// TIA Portal V20 program export: 15 tag tables, 106 data types, 49 data blocks, 136 code blocks (in call order from the OBs), 146 instance data blocks

VAR_GLOBAL   // PLC tag table "Analog_Inputs"
   AI_LaserPowerMeter AT %IW412 : Word;
   AI_AxisB_ClampingPart AT %IW414 : Word;
   AI_LaserAirPressureProcess AT %IW416 : Word;
   AI_InletAirPressure AT %IW418 : Word;
   AI_AmbiantTemperature AT %IW428 : Word;
   AI_MachineTemperature AT %IW430 : Word;
   AI_ColdWaterTemperatureInput AT %IW432 : Word;
   AI_ColdWaterTemperatureOutput AT %IW434 : Word;
   AI_X_AxisTemperaturePT1000 AT %IW436 : Word;
   AI_Y_AxisTemperaturePT1000 AT %IW438 : Word;
   "AI_X_ AxisTemperaturePTC" AT %IW440 : Word;
   "AI_Y_ AxisTemperaturePTC" AT %IW442 : Word;
   AI_NozzleOverpressure AT %IW444 : Word;
   AI_OpticalPathOverpressure AT %IW446 : Word;
   AI_LaserHeadOverpressure AT %IW448 : Word;
   AI_ZL_AxisOverpressure AT %IW450 : Word;
   AI_XY_AxisOverpressure AT %IW452 : Word;
   AI_LeftAspiration AT %IW454 : Word;
   AI_RightAspiration AT %IW456 : Word;
   AI_FreeIW458 AT %IW458 : Word;
   AI_ClimTemperature AT %IW480 : Word;
   AI_FreeIW482 AT %IW482 : Word;
   AI_FreeIW484 AT %IW484 : Word;
   AI_FreeIW486 AT %IW486 : Word;
   AI_SensorControllerStation1 AT %IW460 : Word;
   AI_CabinetTemperature AT %IW462 : Word;
   AI_FreeIW464 AT %IW464 : Word;
   AI_FreeIW466 AT %IW466 : Word;
END_VAR

VAR_GLOBAL   // PLC tag table "Analog_Outputs"
   AQ_NozzleOverpressureSetPoint AT %QW428 : Word;
   AQ_FreeQW482 AT %QW430 : Word;
   AQ_VentilatorSetPoint AT %QW432 : Word;
   AQ_PropValveClimSetPoint AT %QW434 : Word;
END_VAR

VAR_GLOBAL   // PLC tag table "BW_Inputs"
   AI_LifeFlag AT %IW500 : Int;
   DI_JobDone AT %I502.0 : Bool;
   DI_LockShuttle AT %I504.0 : Bool;
   AI_DataSend AT %IW506 : Int;
   AI_DataReceive AT %IW508 : Int;
   DI_NoEmergencyStopAtBwLoader AT %I510.0 : Bool;
   DI_SafetyDoorsClosedAtBwLoader AT %I512.0 : Bool;
   AI_BwInErrorState AT %IW514 : Int;
   DI_UndrilledPartControl AT %I516.0 : Bool;
   DI_DrilledPartControl AT %I518.0 : Bool;
   DI_BackwallControl AT %I520.0 : Bool;
   DI_BwLoaderInSafePos AT %I522.0 : Bool;
   DI_SemiAutoValid AT %I562.0 : Bool;
END_VAR

VAR_GLOBAL   // PLC tag table "BW_Output"
   AQ_LifeFlag AT %QW500 : Int;
   DQ_LoaderRequest AT %Q502.0 : Bool;
   DQ_LockShuttle AT %Q504.0 : Bool;
   AQ_DataSend AT %QW506 : Int;
   AQ_DataReceive AT %QW508 : Int;
   DQ_NoEmergencyStopAtFemto AT %Q510.0 : Bool;
   DQ_SafetyDoorsClosedAtFemto AT %Q512.0 : Bool;
   AQ_FemtoInErrorState AT %QW514 : Int;
   DQ_AutoMode AT %Q516.0 : Bool;
   DQ_JogMode AT %Q518.0 : Bool;
   DQ_GotoSafePos AT %Q520.0 : Bool;
   AQ_Reset AT %QW526 : Int;
   DQ_Emptying AT %Q522.0 : Bool;
   DQ_BW_CtrlInProgress AT %Q524.0 : Bool;
END_VAR

VAR_GLOBAL   // PLC tag table "Cognex"
   ASTriggerReady AT %I690.0 : Bool;   // Acquisition status
   ASTriggerAck AT %I690.1 : Bool;   // Acquisition status
   ASAcquiring AT %I690.2 : Bool;   // Acquisition status
   ASMissedTrig AT %I690.3 : Bool;   // Acquisition status
   ASOfflineResBit1 AT %I690.4 : Bool;   // Acquisition status
   ASOfflineResBit2 AT %I690.5 : Bool;   // Acquisition status
   ASOfflineResBit3 AT %I690.6 : Bool;   // Acquisition status
   ASOnline AT %I690.7 : Bool;   // Acquisition status
   ASAcquiNum AT %IW691 : Word;   // Acquisition status
   ISInspecting AT %I693.0 : Bool;   // Inspection status
   ISToggleInspectDone AT %I693.1 : Bool;   // Inspection status
   ISBufferOverrun AT %I693.2 : Bool;   // Inspection status
   ISResultsValid AT %I693.3 : Bool;   // Inspection status
   ISJobLoading AT %I693.4 : Bool;   // Inspection status
   ISJobLoadComplete AT %I693.5 : Bool;   // Inspection status
   ISJobLoadFailed AT %I693.6 : Bool;   // Inspection status
   ISSetUserDataACk AT %I693.7 : Bool;   // Inspection status
   ISJobPass AT %I694.0 : Bool;   // Inspection status
   SEC0Ack AT %I699.0 : Bool;   // Soft event control
   SEC1Ack AT %I699.1 : Bool;   // Soft event control
   SEC2Ack AT %I699.2 : Bool;   // Soft event control
   SEC3Ack AT %I699.3 : Bool;   // Soft event control
   SEC4Ack AT %I699.4 : Bool;   // Soft event control
   SEC5Ack AT %I699.5 : Bool;   // Soft event control
   SEC6Ack AT %I699.6 : Bool;   // Soft event control
   SEC7Ack AT %I699.7 : Bool;   // Soft event control
   JCJobID AT %IW697 : Word;   // Job control
   IRInspectionID AT %IW600 : Word;   // Inspection result
   IRInspectResultCode AT %IW602 : Word;   // Inspection result
   IRActHoleNrResult AT %IB606 : Byte;   // Inspection result
   ResultDataFromCognex0 AT %ID604 : DWord;
   ResultDataFromCognex1 AT %ID608 : DWord;
   ResultDataFromCognex2 AT %ID612 : DWord;
   ResultDataFromCognex3 AT %ID616 : DWord;
   ACTriggerEnable AT %Q690.0 : Bool;   // Acquisition control
   ACTrigger AT %Q690.1 : Bool;   // Acquisition control
   ACClearAcquirCompl AT %Q690.2 : Bool;   // Acquisition control
   ACSetOffline AT %Q690.7 : Bool;   // Acquisition control
   ICBufferResultsEn AT %Q691.0 : Bool;   // Inspection control
   ICInspectResultsAck AT %Q691.1 : Bool;   // Inspection control
   ICSetUserData AT %Q691.2 : Bool;   // Inspection control
   ICExecuteCmd AT %Q691.3 : Bool;   // Inspection control
   CCSetJobID AT %QW697 : Word;   // Command control
   SEC0 AT %Q699.0 : Bool;   // Soft event control
   SEC1 AT %Q699.1 : Bool;   // Soft event control
   SEC2 AT %Q699.2 : Bool;   // Soft event control
   SEC3 AT %Q699.3 : Bool;   // Soft event control
   SEC4 AT %Q699.4 : Bool;   // Soft event control
   SEC5 AT %Q699.5 : Bool;   // Soft event control
   SEC6 AT %Q699.6 : Bool;   // Soft event control
   SEC7 AT %Q699.7 : Bool;   // Soft event control
   UserDataToCognex0 AT %QD600 : DWord;
   UserDataToCognex1 AT %QD604 : DWord;
   UserDataToCognex2 AT %QD608 : DWord;
   UserDataToCognex3 AT %QD612 : DWord;
   UserDataToCognex4 AT %QD616 : DWord;
   UserDataToCognex5 AT %QD620 : DWord;
   UserDataToCognex6 AT %QD624 : DWord;
   UserDataToCognex7 AT %QD628 : DWord;
END_VAR

VAR_GLOBAL   // PLC tag table "Default tag table"
   System_Byte AT %MB1 : Byte;
   FirstScan AT %M1.0 : Bool;
   DiagStatusUpdate AT %M1.1 : Bool;
   AlwaysTRUE AT %M1.2 : Bool;
   AlwaysFALSE AT %M1.3 : Bool;
   Clock_Byte AT %MB0 : Byte;
   Clock_10Hz AT %M0.0 : Bool;
   Clock_5Hz AT %M0.1 : Bool;
   "Clock_2.5Hz" AT %M0.2 : Bool;
   Clock_2Hz AT %M0.3 : Bool;
   "Clock_1.25Hz" AT %M0.4 : Bool;
   Clock_1Hz AT %M0.5 : Bool;
   "Clock_0.625Hz" AT %M0.6 : Bool;
   "Clock_0.5Hz" AT %M0.7 : Bool;
   Tag_1 AT %M99.0 : Bool;
   Tag_2 AT %MD1000 : DWord;
   Tag_3 AT %MW20 : Word;
   Tag_4 AT %MW40 : Word;
   Tag_5 AT %MW42 : Word;
   Tag_6 AT %MW44 : Word;
   Tag_7 AT %MW100 : Word;
   Tag_8 AT %MW102 : Word;
   Tag_9 AT %MW104 : Word;
   Tag_10 AT %MD150 : DWord;
END_VAR

VAR_GLOBAL   // PLC tag table "Digital_Inputs"
   DI_FreeI0_0 AT %I0.0 : Bool;
   DI_X_AxisBrakePressCtrl AT %I0.1 : Bool;
   DI_Y_AxisBrakePressCtrl AT %I0.2 : Bool;
   DI_BreakerCtrl AT %I0.3 : Bool;
   DI_CabinetTemperatureCtrl AT %I0.4 : Bool;
   DI_UPS_PowerFailure AT %I0.5 : Bool;
   DI_AirPressureCtrl AT %I0.6 : Bool;
   DI_ShutterClosed AT %I0.7 : Bool;
   DI_AirDryerOK AT %I1.0 : Bool;
   DI_UPS_BatteryOK AT %I1.1 : Bool;
   DI_FrontDoorClosed AT %I1.2 : Bool;
   DI_InfeedReadyOK_Start AT %I1.3 : Bool;
   DI_CoolingOK AT %I1.4 : Bool;
   DI_FreeI1_5 AT %I1.5 : Bool;
   DI_PowerReady AT %I1.6 : Bool;
   DI_AlarmI2T AT %I1.7 : Bool;
   DI_HeadLaserBusy AT %I2.0 : Bool;
   DI_HeadLaserBreaker AT %I2.1 : Bool;
   DI_FrontDoorLocked AT %I2.2 : Bool;
   DI_UPS_CommonAlarm AT %I2.3 : Bool;
   DI_UPS_BatteryLow AT %I2.4 : Bool;
   DI_FreeI2_5 AT %I2.5 : Bool;
   DI_HeadChillerHighPressure AT %I2.6 : Bool;
   DI_HeadChillerWaterTemperature AT %I2.7 : Bool;
   DI_HeadChillerFlow AT %I3.0 : Bool;
   DI_HeadChillerCollectivFault AT %I3.1 : Bool;
   DI_HeadChillerWaterLevel AT %I3.2 : Bool;
   DI_UPSByPassActive AT %I3.3 : Bool;
   DI_HeadChillerAmbiantTemperature AT %I3.4 : Bool;
   DI_FreeI3_5 AT %I3.5 : Bool;
   DI_FreeI3_6 AT %I3.6 : Bool;
   DI_FreeI3_7 AT %I3.7 : Bool;
   DI_LoadClampOpened AT %I4.0 : Bool;
   DI_LoadClampNotClosedWithPart AT %I4.1 : Bool;
   DI_UnloadClampOpened AT %I4.2 : Bool;
   DI_UPS_Fault AT %I4.3 : Bool;
   DI_InternalGateLocked AT %I4.4 : Bool;
   DI_ExternalGateLocked AT %I4.5 : Bool;
   DI_InverterActive AT %I4.6 : Bool;
   DI_UnloadClampNotClosedWithPart AT %I4.7 : Bool;
   DI_FreeI5_0 AT %I5.0 : Bool;
   DI_FreeI5_1 AT %I5.1 : Bool;
   DI_InternalGateOpened AT %I5.2 : Bool;
   DI_ExternalGateOpened AT %I5.3 : Bool;
   DI_PowerMeterBackCtrl AT %I5.4 : Bool;
   DI_PowerMeterFrontCtrl AT %I5.5 : Bool;
   DI_FreeI5_6 AT %I5.6 : Bool;
   DI_FreeI5_7 AT %I5.7 : Bool;
   DI_HeadChillerCutOff AT %I6.0 : Bool;
   DI_HeadChillerTemperature AT %I6.1 : Bool;
   DI_FreeI6_2 AT %I6.2 : Bool;
   DI_FreeI6_3 AT %I6.3 : Bool;
   DI_ClampingOpenCtrl AT %I6.4 : Bool;
   DI_B_AxisBrakeReleasedCtrl AT %I6.5 : Bool;
   "DI_FreeI6.6" AT %I6.6 : Bool;
   DI_B_AxisReferencePoint AT %I6.7 : Bool;
   DI_SourceChillerHighPressure AT %I7.0 : Bool;
   DI_SourceChillerWaterTemperature AT %I7.1 : Bool;
   DI_SourceChillerFlow AT %I7.2 : Bool;
   DI_SourceChillerCollectivFault AT %I7.3 : Bool;
   DI_SourceChillerWaterLevel AT %I7.4 : Bool;
   DI_SourceChillerAmbiantTemperature AT %I7.5 : Bool;
   DI_SourceChillerCutOff AT %I7.6 : Bool;
   DI_SourceChillerTemperature AT %I7.7 : Bool;
END_VAR

VAR_GLOBAL   // PLC tag table "Digital_Outputs"
   DQ_FreeQ0_0 AT %Q0.0 : Bool;
   DQ_OperatingCounter AT %Q0.1 : Bool;
   DQ_GeneralAirValve AT %Q0.2 : Bool;
   DQ_SmartLineDisable AT %Q0.3 : Bool;
   DQ_MachineLight AT %Q0.4 : Bool;
   DQ_MachineLightBack AT %Q0.5 : Bool;
   DQ_LightTowerOrange AT %Q0.6 : Bool;
   DQ_LightTowerRed AT %Q0.7 : Bool;
   DQ_LightTowerBlue AT %Q1.0 : Bool;
   DQ_Light_owerGreen AT %Q1.1 : Bool;
   DQ_LightTowerWhite AT %Q1.2 : Bool;
   DQ_Backlight AT %Q1.3 : Bool;
   DQ_FreeQ1_4 AT %Q1.4 : Bool;
   DQ_InfeedON AT %Q1.5 : Bool;
   DQ_AxisActivation AT %Q1.6 : Bool;
   DQ_BuzzerActivation AT %Q1.7 : Bool;
   DQ_ElbaronPowerON AT %Q2.0 : Bool;
   DQ_ObservationCameraLight AT %Q2.1 : Bool;
   DQ_LaserExternalDoorOpening AT %Q2.2 : Bool;
   DQ_CoolingStart AT %Q2.3 : Bool;
   DQ_X_AxisBrakeActivation AT %Q2.4 : Bool;
   DQ_Y_AxisBrakeActivation AT %Q2.5 : Bool;
   DQ_AxisB_TeachInClampingPart AT %Q2.6 : Bool;
   DQ_EPO_UPS AT %Q2.7 : Bool;
   DQ_HeadLaserStart AT %Q3.0 : Bool;
   DQ_HeadLaserStop AT %Q3.1 : Bool;
   DQ_Axis2_PowerContactor AT %Q3.2 : Bool;
   DQ_GasAssistOn AT %Q3.3 : Bool;
   DQ_SmartLineReset AT %Q3.4 : Bool;
   DQ_XY_AxisPowerContactor AT %Q3.5 : Bool;
   DQ_LaserAirPressureProcess AT %Q3.6 : Bool;
   DQ_Bus60V_PowerContactor AT %Q3.7 : Bool;
   DQ_FreeQ4_0 AT %Q4.0 : Bool;
   DQ_FreeQ4_1 AT %Q4.1 : Bool;
   DQ_FreeQ4_2 AT %Q4.2 : Bool;
   DQ_FreeQ4_3 AT %Q4.3 : Bool;
   DQ_LoadClampClosing AT %Q4.4 : Bool;
   DQ_LoadClampOpening AT %Q4.5 : Bool;
   DQ_UnloadClampClosing AT %Q4.6 : Bool;
   DQ_UnloadClampOpening AT %Q4.7 : Bool;
   DQ_ClampingOpening AT %Q5.0 : Bool;
   DQ_ClampingClosing AT %Q5.1 : Bool;
   DQ_B_AxisBrakeRelease AT %Q5.2 : Bool;
   DQ_Suction AT %Q5.3 : Bool;
   DQ_FreeQ5_4 AT %Q5.4 : Bool;
   DQ_FreeQ5_5 AT %Q5.5 : Bool;
   DQ_FreeQ5_6 AT %Q5.6 : Bool;
   DQ_FreeQ5_7 AT %Q5.7 : Bool;
   DQ_ExternalGateClosing AT %Q8.0 : Bool;
   DQ_ExternalGateOpening AT %Q8.1 : Bool;
   DQ_InternalGateClosing AT %Q8.2 : Bool;
   DQ_InternalGateOpening AT %Q8.3 : Bool;
   DQ_PowerMeterRetract AT %Q8.4 : Bool;
   DQ_PowerMeterAdvance AT %Q8.5 : Bool;
   DQ_Blowing AT %Q8.6 : Bool;   //    {ExternalWritable false}
   DQ_FreeQ8_7 AT %Q8.7 : Bool;
   DQ_FreeQ9_0 AT %Q9.0 : Bool;
   DQ_FreeQ9_1 AT %Q9.1 : Bool;
   DQ_FreeQ9_2 AT %Q9.2 : Bool;
   DQ_FreeQ9_3 AT %Q9.3 : Bool;
   DQ_FreeQ9_4 AT %Q9.4 : Bool;
   DQ_FreeQ9_5 AT %Q9.5 : Bool;
   DQ_FreeQ9_6 AT %Q9.6 : Bool;
   DQ_FreeQ9_7 AT %Q9.7 : Bool;
END_VAR

VAR_GLOBAL   // PLC tag table "F-Digital_Inputs"
   FDI_EStopCh1 AT %I1000.0 : Bool;
   FDI_KeySettingModeCh1 AT %I1000.1 : Bool;
   FDI_KeySettingLaserCh1 AT %I1000.2 : Bool;
   FDI_EStopFeedback AT %I1000.3 : Bool;
   FDI_EStopCh2 AT %I1000.4 : Bool;
   FDI_KeySettingModeCh2 AT %I1000.5 : Bool;
   FDI_KeySettingLaserCh2 AT %I1000.6 : Bool;
   FDI_ExternalFeedback AT %I1000.7 : Bool;
   FDI_ReturnPowerLaser AT %I1008.0 : Bool;
   FDI_MaintenanceDoorClosedCh1 AT %I1008.1 : Bool;
   FDI_FrontDoorClosedCh1 AT %I1008.2 : Bool;
   FDI_EstopPowerLaserCh1 AT %I1008.3 : Bool;
   FDI_ReturnShutterLaser AT %I1008.4 : Bool;
   FDI_MaintenanceDoorClosedCh2 AT %I1008.5 : Bool;
   FDI_FrontDoorClosedCh2 AT %I1008.6 : Bool;
   FDI_EstopPowerLaserCh2 AT %I1008.7 : Bool;
   FDI_RoofLeftDoorClosedCh1 AT %I1016.0 : Bool;
   FDI_LaserKeyON_Ch1 AT %I1016.1 : Bool;
   FDI_LaserExternalDoorClosedCh1 AT %I1016.2 : Bool;
   FDI_IntOrExtSasGatesClosedCh1 AT %I1016.3 : Bool;
   FDI_RoofLeftDoorClosedCh2 AT %I1016.4 : Bool;
   FDI_LaserKeyON_Ch2 AT %I1016.5 : Bool;
   FDI_LaserExternalDoorClosedCh2 AT %I1016.6 : Bool;
   FDI_IntOrExtSasGatesClosedCh2 AT %I1016.7 : Bool;
   FDI_BW_LoaderDoorClosedCh1 AT %I1024.0 : Bool;
   FDI_RoofRightDoorClosedCh1 AT %I1024.1 : Bool;
   FDI_SonplasEstopCh1 AT %I1024.2 : Bool;
   FDI_BW_LoaderEStopCh1 AT %I1024.3 : Bool;
   FDI_BW_LoaderDoorClosedCh2 AT %I1024.4 : Bool;
   FDI_RoofRightDoorClosedCh2 AT %I1024.5 : Bool;
   FDI_SonplasEstopCh2 AT %I1024.6 : Bool;
   FDI_BW_LoaderEStopCh2 AT %I1024.7 : Bool;
   FDI_SonplasDoorClosedCh1 AT %I1032.0 : Bool;
   FDI_FreeI1032_1 AT %I1032.1 : Bool;
   FDI_FreeI1032_2 AT %I1032.2 : Bool;
   FDI_FreeI1032_3 AT %I1032.3 : Bool;
   FDI_SonplasDoorClosedCh2 AT %I1032.4 : Bool;
   FDI_FreeI1032_5 AT %I1032.5 : Bool;
   FDI_FreeI1032_6 AT %I1032.6 : Bool;
   FDI_DoorClosedFeedback AT %I1032.7 : Bool;
END_VAR

VAR_GLOBAL   // PLC tag table "F-Digital_Outputs"
   FDQ_StopContactor AT %Q1200.0 : Bool;
   FDQ_LaserContactor AT %Q1200.1 : Bool;
   FDQ_LaserValidation AT %Q1200.2 : Bool;
   FDQ_FrontDoorLock AT %Q1200.3 : Bool;
   FDQ_BW_LoaderEstopRelay AT %Q1206.0 : Bool;
   FDQ_SonplasDoorClosedRelay AT %Q1206.1 : Bool;
   FDQ_FreeQ1206_2 AT %Q1206.2 : Bool;
   FDQ_FreeQ1206_3 AT %Q1206.3 : Bool;
END_VAR

VAR_GLOBAL   // PLC tag table "MCP"
   DI_PB_StartCycle AT %I128.0 : Bool;
   DI_PB_ResetAlarm AT %I128.1 : Bool;
   DI_PB_PowerOFF AT %I128.2 : Bool;
   DI_PB_ShutdownPC AT %I128.3 : Bool;
   DI_PB_LightTest AT %I128.4 : Bool;
   DI_PB_RemoteOpenShutter AT %I128.6 : Bool;
   DI_FreeI128_7 AT %I128.7 : Bool;
   DQ_AlarmBlueLED AT %Q127.1 : Bool;
   DQ_StartCycleGreenLED AT %Q127.0 : Bool;
   DQ_RemoteOpenShutterWhiteLED AT %Q127.5 : Bool;
   DQ_ShutdownPCYellowLED AT %Q127.3 : Bool;
   DQ_LightTestWhiteLED AT %Q127.4 : Bool;
   DI_PB_PowerON AT %I128.5 : Bool;
   DQ_PowerOnGreenLED AT %Q127.2 : Bool;
   DQ_FreeQ127_6 AT %Q127.6 : Bool;
   DQ_FreeQ127_7 AT %Q127.7 : Bool;
   MCP1_In AT %I118.0 : "LBP_typeMcp483StandardInput";
   MCP1_Out AT %Q120.0 : "LBP_typeMcp483StandardOutput";
END_VAR

VAR_GLOBAL   // PLC tag table "Safety_Drive"
   Axis01_X_Status AT %I6812.0 : "LDrvSafe_typeSinaTlg903Status";
   Axis02_Y_Status AT %I6828.0 : "LDrvSafe_typeSinaTlg903Status";
   Axis03_ZM_Status AT %I6844.0 : "LDrvSafe_typeSinaTlg903Status";
   Axis04_B_Status AT %I6764.0 : "LDrvSafe_typeSinaTlg903Status";
   Axis05_U1_Status AT %I6700.0 : "LDrvSafe_typeSinaTlg903Status";
   Axis06_U2_Status AT %I6748.0 : "LDrvSafe_typeSinaTlg903Status";
   Axis07_V_Status AT %I6716.0 : "LDrvSafe_typeSinaTlg903Status";
   Axis08_W_Status AT %I6732.0 : "LDrvSafe_typeSinaTlg903Status";
   Axis09_ZL_Status AT %I6860.0 : "LDrvSafe_typeSinaTlg903Status";
   Axis01_X_Control AT %Q6812.0 : "LDrvSafe_typeSinaTlg903Control";
   Axis02_Y_Control AT %Q6828.0 : "LDrvSafe_typeSinaTlg903Control";
   Axis03_ZM_Control AT %Q6844.0 : "LDrvSafe_typeSinaTlg903Control";
   Axis04_B_Control AT %Q6764.0 : "LDrvSafe_typeSinaTlg903Control";
   Axis05_U1_Control AT %Q6700.0 : "LDrvSafe_typeSinaTlg903Control";
   Axis06_U2_Control AT %Q6748.0 : "LDrvSafe_typeSinaTlg903Control";
   Axis07_V_Control AT %Q6716.0 : "LDrvSafe_typeSinaTlg903Control";
   Axis08_W_Control AT %Q6732.0 : "LDrvSafe_typeSinaTlg903Control";
   Axis09_ZL_Control AT %Q6860.0 : "LDrvSafe_typeSinaTlg903Control";
END_VAR

VAR_GLOBAL   // PLC tag table "Sonplas_Inputs"
   DI_SonplasDiagDPCoupler AT %I200.0 : Bool;
   DI_SonplasReady AT %I200.1 : Bool;
   DI_SonplasNoEStop AT %I200.2 : Bool;
   DI_SonplasDoorsClosed AT %I200.3 : Bool;
   DI_SonplasRunError AT %I200.4 : Bool;
   DI_SonplasFreeI200_5 AT %I200.5 : Bool;
   DI_SonplasFreeI200_6 AT %I200.6 : Bool;
   DI_SonplasFreeI200_7 AT %I200.7 : Bool;
   DI_SonplasFreeI201_0 AT %I201.0 : Bool;
   DI_SonplasOutCollision AT %I201.1 : Bool;
   DI_SonplasFreeI201_2 AT %I201.2 : Bool;
   DI_SonplasFreeI201_3 AT %I201.3 : Bool;
   DI_SonplasFreeI201_4 AT %I201.4 : Bool;
   DI_SonplasFreeI201_5 AT %I201.5 : Bool;
   DI_SonplasFreeI201_6 AT %I201.6 : Bool;
   DI_SonplasFreeI201_7 AT %I201.7 : Bool;
   DI_SonplasShuttle1Finished AT %I202.0 : Bool;
   DI_SonplasFreeI202_1 AT %I202.1 : Bool;
   DI_SonplasFreeI202_2 AT %I202.2 : Bool;
   DI_SonplasFreeI202_3 AT %I202.3 : Bool;
   DI_SonplasFreeI202_4 AT %I202.4 : Bool;
   DI_SonplasFreeI202_5 AT %I202.5 : Bool;
   DI_SonplasFreeI202_6 AT %I202.6 : Bool;
   DI_SonplasFreeI202_7 AT %I202.7 : Bool;
   DI_SonplasShuttle2Finished AT %I203.0 : Bool;
   DI_SonplasFreeI203_1 AT %I203.1 : Bool;
   DI_SonplasFreeI203_2 AT %I203.2 : Bool;
   DI_SonplasFreeI203_3 AT %I203.3 : Bool;
   DI_SonplasFreeI203_4 AT %I203.4 : Bool;
   DI_SonplasFreeI203_5 AT %I203.5 : Bool;
   DI_SonplasFreeI203_6 AT %I203.6 : Bool;
   DI_SonplasFreeI203_7 AT %I203.7 : Bool;
   DI_SonplasFlowResultAvail AT %I244.0 : Bool;
   DI_SonplasFreeI244_1 AT %I244.1 : Bool;
   DI_SonplasFreeI244_2 AT %I244.2 : Bool;
   DI_SonplasFreeI244_3 AT %I244.3 : Bool;
   DI_SonplasFreeI244_4 AT %I244.4 : Bool;
   DI_SonplasFreeI244_5 AT %I244.5 : Bool;
   DI_SonplasFreeI244_6 AT %I244.6 : Bool;
   DI_SonplasFreeI244_7 AT %I244.7 : Bool;
   AI_SonplasDMC_Code1 AT %IB204 : Byte;
   AI_SonplasDMC_Code2 AT %IB224 : Byte;
   AI_SonplasFlowResult AT %IW245 : Word;
   AI_SonplasDMC_CodeFlow AT %IB247 : Byte;
END_VAR

VAR_GLOBAL   // PLC tag table "Sonplas_Outputs"
   DQ_SonplasDiagDPCoupler AT %Q200.0 : Bool;
   DQ_SonplasReady AT %Q200.1 : Bool;
   DQ_SonplasNoEStop AT %Q200.2 : Bool;
   DQ_SonplasDoorsClosed AT %Q200.3 : Bool;
   DQ_SonplasRunError AT %Q200.4 : Bool;
   DQ_SonplasFreeQ200_5 AT %Q200.5 : Bool;
   DQ_SonplasFreeQ200_6 AT %Q200.6 : Bool;
   DQ_SonplasFreeQ200_7 AT %Q200.7 : Bool;
   DQ_SonplasFreeQ201_0 AT %Q201.0 : Bool;
   DQ_SonplasFreeQ201_1 AT %Q201.1 : Bool;
   DQ_SonplasFreeQ201_2 AT %Q201.2 : Bool;
   DQ_SonplasFreeQ201_3 AT %Q201.3 : Bool;
   DQ_SonplasFreeQ201_4 AT %Q201.4 : Bool;
   DQ_SonplasFreeQ201_5 AT %Q201.5 : Bool;
   DQ_SonplasFreeQ201_6 AT %Q201.6 : Bool;
   DQ_SonplasFreeQ201_7 AT %Q201.7 : Bool;
   DQ_SonplasShuttle1InPos AT %Q202.0 : Bool;
   DQ_SonplasFreeQ202_1 AT %Q202.1 : Bool;
   DQ_SonplasFreeQ202_2 AT %Q202.2 : Bool;
   DQ_SonplasFreeQ202_3 AT %Q202.3 : Bool;
   DQ_SonplasFreeQ202_4 AT %Q202.4 : Bool;
   DQ_SonplasFreeQ202_5 AT %Q202.5 : Bool;
   DQ_SonplasPart1OK AT %Q202.6 : Bool;
   DQ_SonplasPart1NOK AT %Q202.7 : Bool;
   DQ_SonplasShuttle2InPos AT %Q203.0 : Bool;
   DQ_SonplasFreeQ203_1 AT %Q203.1 : Bool;
   DQ_SonplasFreeQ203_2 AT %Q203.2 : Bool;
   DQ_SonplasFreeQ203_3 AT %Q203.3 : Bool;
   DQ_SonplasFreeQ203_4 AT %Q203.4 : Bool;
   DQ_SonplasFreeQ203_5 AT %Q203.5 : Bool;
   DQ_SonplasPart2OK AT %Q203.6 : Bool;
   DQ_SonplasPart2NOK AT %Q203.7 : Bool;
   DQ_SonplasResultAccepted AT %Q244.0 : Bool;
   DQ_SonplasFreeQ244_1 AT %Q244.1 : Bool;
   DQ_SonplasFreeQ244_2 AT %Q244.2 : Bool;
   DQ_SonplasFreeQ244_3 AT %Q244.3 : Bool;
   DQ_SonplasFreeQ244_4 AT %Q244.4 : Bool;
   DQ_SonplasFreeQ244_5 AT %Q244.5 : Bool;
   DQ_SonplasFreeQ244_6 AT %Q244.6 : Bool;
   DQ_SonplasFreeQ244_7 AT %Q244.7 : Bool;
   AQ_SonplasDMC_Code1 AT %QB204 : Byte;
   AQ_SonplasDMC_Code2 AT %QB224 : Byte;
END_VAR

VAR_GLOBAL   // PLC tag table "UPS"
   M_ShutdownPCRequest AT %MW2 : Int;
   M_ShutdownPCResponse AT %MW4 : Int;
END_VAR

TYPE "UDT_Alarms"
   STRUCT
      Id : DInt;
      Severity : Byte;
      Acknowledge : Bool;
   END_STRUCT;
END_TYPE

TYPE "UDT_AxisPosition"
   STRUCT
      Axis_U : Struct
         PosExternalLoadUnload : Real;
         PosExternalLoadUnloadManu : Real;
         PosPartControl : Real;
         PosBwControl : Real;
         PosInternalLoadUnload : Real;
         PosExtGateExt : Real;
         PosIntGateExt : Real;
         PosExtGateInt : Real;
         PosIntGateInt : Real;
      END_STRUCT;
      Axis_V : Struct
         PosLoadUnload : Real;
         PosSafe : Real;
      END_STRUCT;
      Axis_W : Struct
         PosLoadUnload : Real;
         PosSafe : Real;
         PosApproach : Real;
      END_STRUCT;
   END_STRUCT;
END_TYPE

TYPE "UDT_AxisPosition_OLD"
   STRUCT
      Axis_U : Struct
         PosExternalLoad : Real;
         PosExternalUnload : Real;
         PosSas : Real;
         PosBlowing : Real;
         PosControlUndrilled : Real;
         PosControlDrilled : Real;
         PosInternalLoadUndrilled : Real;
         PosInternalUnloadDrilled : Real;
         PosSemiAuto : Real;
         PosExtGateExt : Real;
         PosIntGateExt : Real;
         PosExtGateInt : Real;
         PosIntGateInt : Real;
      END_STRUCT;
      Axis_V : Struct
         PosShuttleUndrilled : Real;
         PosShuttleDrilled : Real;
         PosWashingVacuum : Real;
         PosWashingBrush : Real;
         PosHome : Real;
         PosChangeBackwall : Real;
      END_STRUCT;
      Axis_W : Struct
         PosUp : Real;
         PosShuttleUndrilled : Real;
         PosShuttleDrilled : Real;
         PosWashingVacuum : Real;
         PosWashingBrush : Real;
         PosChangeBackwall : Real;
      END_STRUCT;
      Axis_X : Struct
         PosChangeBackwall : Real;
      END_STRUCT;
      Axis_Y : Struct
         PosChangeBackwall : Real;
      END_STRUCT;
      Axis_ZM : Struct
         PosChangeBackwall : Real;
      END_STRUCT;
      Axis_ZL : Struct
         PosChangeBackwall : Real;
      END_STRUCT;
      Axis_B : Struct
         PosChangeBackwall : Real;
      END_STRUCT;
      Axis_C : Struct
         PosChangeBackwall : Real;
      END_STRUCT;
   END_STRUCT;
END_TYPE

TYPE "UDT_BoolEnable"
   STRUCT
      IsEnabled : Bool;
      Value : Bool;
   END_STRUCT;
END_TYPE

TYPE "UDT_FormatMsg"
   STRUCT
      Id : DInt;
      Severity : Byte;
      Active : Bool;
   END_STRUCT;
END_TYPE

TYPE "UDT_MaintenanceElement"
   STRUCT
      RunTime : Real;   // Temps de fonctionnement actuel (en unité de temps)
      RunTimeSec : Real;   // Temps de fonctionnement actuel (en secondes)
      WarningThreshold : Int;   // Seuil d'avertissement en % (par défaut 80%)
      AlarmThreshold : Int;   // Durée maximale avant maintenance
      TimeUnit : Int;   // Unité de temps (0:Minutes, 1:Hours, 2:Days)
      ResetRunTime : Bool;   // Reset Temps de fonctionnement actuel
   END_STRUCT;
END_TYPE

TYPE "UDT_Msg"
   STRUCT
      ID : Int;
      Number : DInt;
      Active : Bool;
      Level : Int;
   END_STRUCT;
END_TYPE

TYPE "UDT_POS_AXES_UVW"
   STRUCT
      U_POS_EXTERNAL_LOAD : Real;
      U_POS_EXTERNAL_UNLOAD : Real;
      U_POS_SAS : Real;
      U_POS_BLOWING : Real;
      U_POS_DETECTOR_LOAD : Real;
      U_POS_DETECTOR_UNLOAD : Real;
      U_POS_INTERNAL_LOADER_LOAD : Real;
      U_POS_INTERNAL_LOADER_UNLOAD : Real;
      U_POS_OUT_INTERNAL_LOADER : Real;
      U_DELTA_POS_INTERN_LOADER_LOAD_UNLOAD : Real;
      U_POS_SEMI_AUTO : Real;
      V_POS_SHUTTLE_LOAD : Real;
      V_POS_SHUTTLE_UNLOAD : Real;
      V_POS_WASHING : Real;
      W_POS_UP : Real;
      W_POS_SHUTTLE_LOAD : Real;
      W_POS_SHUTTLE_UNLOAD : Real;
      W_POS_WASHING : Real;
      X_POS_CHANGE_BW : Real;
      Y_POS_CHANGE_BW : Real;
   END_STRUCT;
END_TYPE

TYPE "UDT_PowermeterMeasure"
   STRUCT
      NbMeasure : Int := 100;
      ActualMeasure : Int;
      ActualTotalMeas : Real;
      Table_full : Bool;   // TRUE when the table are fully of measures
      Measures : Array[0..99] of Struct
         Time_day : Time_Of_Day;
         Day_meas : Date;
         Job_meas : Int;
         ValuePower : Real;
         ValueCM : Real;
      END_STRUCT;
   END_STRUCT;
END_TYPE

TYPE "UDT_SequenceInterface"
   STRUCT
      Error : Bool;
      Reset : Bool;
      SequenceReleased : Bool;
      SequenceRun : Bool;
      JobDone : Bool;
      StartRequest : Bool;
   END_STRUCT;
END_TYPE

TYPE "UDT_Token_GUD"
   STRUCT
      Syntax_ID { ExternalAccessible := 'False'; ExternalVisible := 'False'; ExternalWritable := 'False'} : Byte;
      Area_unit { ExternalAccessible := 'False'; ExternalVisible := 'False'; ExternalWritable := 'False'} : Byte;
      Col_index { ExternalAccessible := 'False'; ExternalVisible := 'False'; ExternalWritable := 'False'} : Word;
      Line_index { ExternalAccessible := 'False'; ExternalVisible := 'False'; ExternalWritable := 'False'} : Word;
      Block_type { ExternalAccessible := 'False'; ExternalVisible := 'False'; ExternalWritable := 'False'} : Byte;
      Num_lines { ExternalAccessible := 'False'; ExternalVisible := 'False'; ExternalWritable := 'False'} : Byte;
      S7_type { ExternalAccessible := 'False'; ExternalVisible := 'False'; ExternalWritable := 'False'} : Byte;
      Nc_length { ExternalAccessible := 'False'; ExternalVisible := 'False'; ExternalWritable := 'False'} : Byte;
   END_STRUCT;
END_TYPE

TYPE "UDT_EmptyPosition"
   STRUCT
      Presence : "UDT_PartPresence";
      States : "UDT_PartStates";
   END_STRUCT;
END_TYPE

TYPE "UDT_Holes"
   STRUCT
      Pos_X { ExternalAccessible := 'False'; ExternalVisible := 'False'; ExternalWritable := 'False'} : Real := 999.99;
      Pos_Y { ExternalAccessible := 'False'; ExternalVisible := 'False'; ExternalWritable := 'False'} : Real := 999.99;
      Pos_Z { ExternalAccessible := 'False'; ExternalVisible := 'False'; ExternalWritable := 'False'} : Real := 999.99;
      Pos_RX { ExternalAccessible := 'False'; ExternalVisible := 'False'; ExternalWritable := 'False'} : Real := 999.99;
      Pos_RY { ExternalAccessible := 'False'; ExternalVisible := 'False'; ExternalWritable := 'False'} : Real := 999.99;
      Pos_RZ { ExternalAccessible := 'False'; ExternalVisible := 'False'; ExternalWritable := 'False'} : Real := 999.99;
      Pos_delta_RX { ExternalAccessible := 'False'; ExternalVisible := 'False'; ExternalWritable := 'False'} : Real := 999.99;
      Pos_delta_RY { ExternalAccessible := 'False'; ExternalVisible := 'False'; ExternalWritable := 'False'} : Real := 999.99;
      Pos_delta_RZ { ExternalAccessible := 'False'; ExternalVisible := 'False'; ExternalWritable := 'False'} : Real := 999.99;
      Measure_X { ExternalAccessible := 'False'; ExternalVisible := 'False'; ExternalWritable := 'False'} : Real := 999.99;
      Measure_Y { ExternalAccessible := 'False'; ExternalVisible := 'False'; ExternalWritable := 'False'} : Real := 999.99;
      Measure_Z { ExternalAccessible := 'False'; ExternalVisible := 'False'; ExternalWritable := 'False'} : Real := 999.99;
      Measure_D { ExternalAccessible := 'False'; ExternalVisible := 'False'; ExternalWritable := 'False'} : Real := 999.99;
      Measure_concentricity_before { ExternalAccessible := 'False'; ExternalVisible := 'False'; ExternalWritable := 'False'} : Real := 999.99;
      Measure_concentricity_after { ExternalAccessible := 'False'; ExternalVisible := 'False'; ExternalWritable := 'False'} : Real := 999.99;
      Job_laser { ExternalAccessible := 'False'; ExternalVisible := 'False'; ExternalWritable := 'False'} : Int := 999;
   END_STRUCT;
END_TYPE

TYPE "UDT_PartPosition"
   STRUCT
      Undrilled : Struct
         Presence : "UDT_PartPresence";
         States : "UDT_PartStates";
      END_STRUCT;
      Drilled : Struct
         Presence : "UDT_PartPresence";
         States : "UDT_PartStates";
      END_STRUCT;
   END_STRUCT;
END_TYPE

TYPE "UDT_PartPresence"
   STRUCT
      Part : Bool;
      BW : Bool;
   END_STRUCT;
END_TYPE

TYPE "UDT_PartState"
   STRUCT
      Good : Bool;
      Unknown : Bool;
      Bad : Bool;
      Absent : Bool;
      PresentUnexpected : Bool;
      AbsentUnexpected : Bool;
   END_STRUCT;
END_TYPE

TYPE "UDT_PartStates"
   STRUCT
      BW : Struct
         Good : Bool;
         Unknown : Bool;
         Bad : Bool;
         Absent : Bool;
         PresentUnexpected : Bool;
         AbsentUnexpected : Bool;
      END_STRUCT;
      Part : Struct
         Good : Bool;
         Unknown : Bool;
         Bad : Bool;
         Absent : Bool;
         PresentUnexpected : Bool;
         AbsentUnexpected : Bool;
      END_STRUCT;
   END_STRUCT;
END_TYPE

TYPE "UDT_Tracability"
   STRUCT
      Part_id { ExternalAccessible := 'False'; ExternalVisible := 'False'; ExternalWritable := 'False'} : Int;
      Status { ExternalAccessible := 'False'; ExternalVisible := 'False'; ExternalWritable := 'False'} : Int;
      FailCode { ExternalAccessible := 'False'; ExternalVisible := 'False'; ExternalWritable := 'False'} : Int;
      FailCodeBackwall { ExternalAccessible := 'False'; ExternalVisible := 'False'; ExternalWritable := 'False'} : Int;
      DMC { ExternalAccessible := 'False'; ExternalVisible := 'False'; ExternalWritable := 'False'} : Array[0..19] of Byte;
      OrderNbr { ExternalAccessible := 'False'; ExternalVisible := 'False'; ExternalWritable := 'False'} : String[64];
      IdentNbr { ExternalAccessible := 'False'; ExternalVisible := 'False'; ExternalWritable := 'False'} : String[64];
      BatchNbr { ExternalAccessible := 'False'; ExternalVisible := 'False'; ExternalWritable := 'False'} : String[64];
      OperatorNbr { ExternalAccessible := 'False'; ExternalVisible := 'False'; ExternalWritable := 'False'} : String[64];
      Comment { ExternalAccessible := 'False'; ExternalVisible := 'False'; ExternalWritable := 'False'} : String[192];
      WOZ_Status : Int;
      WOC_Status : Int;
      WOZ_Measure { ExternalAccessible := 'False'; ExternalVisible := 'False'; ExternalWritable := 'False'} : Real;
      WOC_Measure { ExternalAccessible := 'False'; ExternalVisible := 'False'; ExternalWritable := 'False'} : Real;
      TotalCycleTime { ExternalAccessible := 'False'; ExternalVisible := 'False'; ExternalWritable := 'False'} : Int;
      LaserCycleTime { ExternalAccessible := 'False'; ExternalVisible := 'False'; ExternalWritable := 'False'} : Int;
      MeasureLoadCycleTime { ExternalAccessible := 'False'; ExternalVisible := 'False'; ExternalWritable := 'False'} : Int;
      FlowResult : Real;
      HoleSettings { ExternalAccessible := 'False'; ExternalVisible := 'False'; ExternalWritable := 'False'} : Array[0..99] of "UDT_Holes";
   END_STRUCT;
END_TYPE

TYPE "UDT_Tracability_Data"
   STRUCT
      Nb_of_Records { ExternalAccessible := 'False'; ExternalVisible := 'False'; ExternalWritable := 'False'} : Int := 100;
      Nb_of_Holes { ExternalAccessible := 'False'; ExternalVisible := 'False'; ExternalWritable := 'False'} : Int := 100;
      STRUCT_PART { ExternalAccessible := 'False'; ExternalVisible := 'False'; ExternalWritable := 'False'} : Array[0..99] of Struct
         Part_id : Int;
         Status : Int;
         Fail_code : Int;
         Raw_type : Int;
         Workpiece_holder_type : Int;
         Workpiece_holder_Nbr : Int;
         Datamatrix_code : Array[0..19] of Byte;
         Order_nbr : String[64];
         Ident_nbr : String[64];
         Batch_nbr : String[64];
         Operator_nbr : String[64];
         Comment : String[192];
         WOZ : Real;
         WOC : Real;
         Total_cycle_time : Int;
         Laser_cycle_time : Int;
         Measure_load_cycle_time : Int;
         STRUCT_HOLE : Array[0..99] of "UDT_Holes";
      END_STRUCT;
   END_STRUCT;
   // STRUCT_PART[1..10].Part_id := -1;
END_TYPE

TYPE "UDT_MaintenanceTask"
   STRUCT
      Elapsed : Bool;
      Id : Bool;
      Period : Bool;
      Warning : Bool;
   END_STRUCT;
END_TYPE

TYPE "UDT_OPCButtons"
   STRUCT
      bBlink : Bool;   // From PLC
      bClick : Bool;   // From HMI
      bEnable : Bool;   // From PLC
      bIsPressed : Bool;   // From PLC
      eColor : Int;   // From PLC
   END_STRUCT;
END_TYPE

TYPE "AnalogInAction_DT"
   STRUCT
      BadPartOnFixture { ExternalVisible := 'False'} : Bool;
      ID_Measure : Int;
   END_STRUCT;
END_TYPE

TYPE "AnalogInDataHMI_DT"
   STRUCT
      ID_Measure : Int;
      CurrentValue : Real;
      TargetValue : Real;
      ThresholdAlarmMin : Real;
      ThresholdWarningMin : Real;
      ThresholdWarningMax : Real;
      ThresholdAlarmMax : Real;
      AxFactor { ExternalAccessible := 'False'; ExternalVisible := 'False'; ExternalWritable := 'False'} : Real := 1.0;   // A Factor Correction type y= Ax + B (A = 1 if no correction)
      BOffset { ExternalAccessible := 'False'; ExternalVisible := 'False'; ExternalWritable := 'False'} : Real;   // B Offset Correction type y= Ax + B (B = 0 if no correction)
      StartTime : Time;
      Update : Bool;
   END_STRUCT;
END_TYPE

TYPE "AnalogInDataPLC_DT"
   STRUCT
      LimitUp { ExternalAccessible := 'False'; ExternalVisible := 'False'; ExternalWritable := 'False'} : Real;   // Limit up real value
      LimitDown { ExternalAccessible := 'False'; ExternalVisible := 'False'; ExternalWritable := 'False'} : Real;   // Limit down real value
      TypeProbe { ExternalAccessible := 'False'; ExternalVisible := 'False'; ExternalWritable := 'False'} : Int;   // 0 : PT100, 1 : PT1000, 2 : 0-10V, 3: -10+10V, 4 : RES600, 5 : SL5201 (0-10V), 6 : PTC
      DelayAlarmMin : Time;
      DelayWarningMin : Time;
      DelayWarningMax : Time;
      DelayAlarmMax : Time;
      EnableAlarmMin : Bool;
      EnableWarningMin : Bool;
      EnableWarningMax : Bool;
      EnableAlarmMax : Bool;
      BadPartOnFixture { ExternalVisible := 'False'} : Bool;
   END_STRUCT;
END_TYPE

TYPE "AnalogInput_DT"
   STRUCT
      SWRealValue : Real;   // Software real value use in PLC
      HWWordValue : Word;   // Hardware value direclty from physical input
   END_STRUCT;
END_TYPE

TYPE "AnalogOutput_DT"
   STRUCT
      SWRealValue : Real;   // Software real value use in PLC
      HWWordValue : Word;   // Hardware value direclty to physical input
   END_STRUCT;
END_TYPE

TYPE "Analog_Ctrl_DT"
   STRUCT
      Type_of_probe { ExternalVisible := 'False'} : Int;   // PT100=0, PT1000=1, NTC=2, RES600=3, 0-10V=4, -10+10V=5, 0-2000=6 / PT100=0(FC71:0, PT1000=1(FC71:1), NTC=2(FC74), RES600=3
      Target_value : Real;
      SWRealValue { ExternalVisible := 'False'} : Real;
      HWWordValue : Word;
      Time_delay { ExternalVisible := 'False'} : Time;
      Threshold_Alarm_min { ExternalVisible := 'False'} : Real;
      Threshold_Warning_min { ExternalVisible := 'False'} : Real;
      Threshold_Warning_max { ExternalVisible := 'False'} : Real;
      Threshold_Alarm_max { ExternalVisible := 'False'} : Real;
      Num_alarm_min { ExternalVisible := 'False'} : Int := -1;
      Num_warning_min { ExternalVisible := 'False'} : Int := -1;
      Num_warning_max { ExternalVisible := 'False'} : Int := -1;
      Num_alarm_max { ExternalVisible := 'False'} : Int := -1;
      Num_alarm_out_of_range { ExternalVisible := 'False'} : Int := -1;
      Stop_machine { ExternalVisible := 'False'} : Bool;
      Bad_part_on_laser { ExternalVisible := 'False'} : Bool;
      axFactor : Real;
      bOffset : Real;
      iLimitUp : Real;
      iLimitDown : Real;
   END_STRUCT;
END_TYPE

TYPE "DigitalInput_DT"
   STRUCT
      SWStatus : Bool;   // Software status use in PLC code
      SWPositiveFront : Bool;   // Positive front of software status
      SWNegativeFront : Bool;   // Negative front of sofware status
      HWStatus : Bool;   // Hardware status directly from physical input
   END_STRUCT;
END_TYPE

TYPE "DigitalOutput_DT"
   STRUCT
      SWStatus : Bool;   // Software status use in PLC code
      HWStatus : Bool;   // Hardware status directly set to physical output
   END_STRUCT;
END_TYPE

TYPE "Temperature_DT"
   STRUCT
      axFactor : Real := 1.0;
      bOffset : Real := 0.0;
   END_STRUCT;
END_TYPE

TYPE "LDrvSafe_typeSinaTlg903Control"
TITLE = LDrvSafe_typeSinaTlg903Control
// Failsafe user-defined data type for PROFIsafe telegram 903 to control the Safety Integrated Functions of SINAMICS
// stored: IsFailsafeCompliant true
   STRUCT
      STO { ExternalWritable := 'False'} : Bool;   // Safety Function Safe Torque Off
      SS1 { ExternalWritable := 'False'} : Bool;   // Safety Function Safe Stop 1
      SS2 { ExternalWritable := 'False'} : Bool;   // Safety Function Safe Stop 2
      SOS { ExternalWritable := 'False'} : Bool;   // Safety Function Safe Operating Stop
      SLS { ExternalWritable := 'False'} : Bool;   // Safety Function Safely-limited Speed
      reserved1 { ExternalWritable := 'False'} : Bool;   // Reserve bit 1
      SLP { ExternalWritable := 'False'} : Bool;   // Safety Function Safely-limited Position
      internalEventAcknowledge { ExternalWritable := 'False'} : Bool;   // Acknowledge Safety errors in the drive
      SLA { ExternalWritable := 'False'} : Bool;   // Safety Function Safely-limited Acceleration
      selectSLSbit0 { ExternalWritable := 'False'} : Bool;   // Select one of the the four SLS limits; operates together with bit 1
      selectSLSbit1 { ExternalWritable := 'False'} : Bool;   // Select one of the the four SLS limits; operates together with bit 0
      reserved3 { ExternalWritable := 'False'} : Bool;   // Reserve bit 3
      SDIpositive { ExternalWritable := 'False'} : Bool;   // Safety Function Safe Direction (positive direction)
      SDInegative { ExternalWritable := 'False'} : Bool;   // Safety Function Safe Direction (negative direction)
      reserved4 { ExternalWritable := 'False'} : Bool;   // Reserve bit 4
      reserved5 { ExternalWritable := 'False'} : Bool;   // Reserve bit 5
      reserved6 { ExternalWritable := 'False'} : Bool;   // Reserve bit 6
      reserved7 { ExternalWritable := 'False'} : Bool;   // Reserve bit 7
      reserved8 { ExternalWritable := 'False'} : Bool;   // Reserve bit 8
      selectSLPrange { ExternalWritable := 'False'} : Bool;   // Select one of the two SLP ranges
      reserved9 { ExternalWritable := 'False'} : Bool;   // Reserve bit 9
      reserved10 { ExternalWritable := 'False'} : Bool;   // Reserve bit 10
      reserved11 { ExternalWritable := 'False'} : Bool;   // Reserve bit 11
      SCA { ExternalWritable := 'False'} : Bool;   // Safety Function Safe Cam
      selectGearboxStageBit0 { ExternalWritable := 'False'} : Bool;   // Select one of the the eight gearbox stages; operates together with bit 1 and 2
      selectGearboxStageBit1 { ExternalWritable := 'False'} : Bool;   // Select one of the the eight gearbox stages; operates together with bit 0 and 2
      selectGearboxStageBit2 { ExternalWritable := 'False'} : Bool;   // Select one of the the eight gearbox stages; operates together with bit 0 and 1
      switchoverGearboxStage { ExternalWritable := 'False'} : Bool;   // Higher position tolerance at gearbox switching
      SS2E { ExternalWritable := 'False'} : Bool;   // Safety Function Safe Stop 2 with external stop
      SS2ESR { ExternalWritable := 'False'} : Bool;   // Safety Function Safe Stop 2 with Extended Stop and Retract
      reserved14 { ExternalWritable := 'False'} : Bool;   // Reserve bit 14
      reserved15 { ExternalWritable := 'False'} : Bool;   // Reserve bit 15
      variableSLS { ExternalWritable := 'False'} : Int;   // SLS limit 1 can be varied within 1 and 32.767 (0.03 and 100%)
   END_STRUCT;
END_TYPE

TYPE "LDrvSafe_typeSinaTlg903Status"
TITLE = LDrvSafe_typeSinaTlg903Status
// Failsafe user-defined data type for PROFIsafe telegram 903 to get status information of Safety Integrated Functions of SINAMICS
// stored: IsFailsafeCompliant true
   STRUCT
      STOactive { ExternalWritable := 'False'} : Bool;   // Safety Function Safe Torque Off active
      SS1active { ExternalWritable := 'False'} : Bool;   // Safety Function Safe Stop 1 active
      SS2active { ExternalWritable := 'False'} : Bool;   // Safety Function Safe Stop 2 active
      SOSactive { ExternalWritable := 'False'} : Bool;   // Safety Function Safe Operating Stop active
      SLSactive { ExternalWritable := 'False'} : Bool;   // Safety Function Safely-limited Speed active
      reserved1 { ExternalWritable := 'False'} : Bool;   // Reserve bit 1
      SLPactive { ExternalWritable := 'False'} : Bool;   // Safety Function Safely-limited Position active
      internalEvent { ExternalWritable := 'False'} : Bool;   // Internal Event occured (Safety error in SINAMICS)
      SLAactive { ExternalWritable := 'False'} : Bool;   // Safety Function Safely-limited Acceleration active
      SLSbit0Active { ExternalWritable := 'False'} : Bool;   // One of the the four SLS limits is active; operates together with bit 1
      SLSbit1Active { ExternalWritable := 'False'} : Bool;   // One of the the four SLS limits is active; operates together with bit 0
      reserved3 { ExternalWritable := 'False'} : Bool;   // Reserve bit 3
      SDIpositiveActive { ExternalWritable := 'False'} : Bool;   // Safety Function Safe Direction (positive direction) active
      SDInegativeActive { ExternalWritable := 'False'} : Bool;   // Safety Function Safe Direction (negative direction) active
      reserved4 { ExternalWritable := 'False'} : Bool;   // Reserve bit 4
      SSMactive { ExternalWritable := 'False'} : Bool;   // Safety Function Safe Speed Monitor; signals, if safe speed is below paramterizable speed limit
      reserved5 { ExternalWritable := 'False'} : Bool;   // Reserve bit 5
      reserved6 { ExternalWritable := 'False'} : Bool;   // Reserve bit 6
      reserved7 { ExternalWritable := 'False'} : Bool;   // Reserve bit 7
      SLPrangeActive { ExternalWritable := 'False'} : Bool;   // SLP position range 1 or 2 is active
      reserved8 { ExternalWritable := 'False'} : Bool;   // Reserve bit 8
      reserved9 { ExternalWritable := 'False'} : Bool;   // Reserve bit 9
      safePositionValid { ExternalWritable := 'False'} : Bool;   // Safe Position is valid
      safelyReferenced { ExternalWritable := 'False'} : Bool;   // Drive is safely referenced
      statusFDI0 { ExternalWritable := 'False'} : Bool;   // Status of Failsafe Digital Input 0
      statusFDI1 { ExternalWritable := 'False'} : Bool;   // Status of Failsafe Digital Input 1
      statusFDI2 { ExternalWritable := 'False'} : Bool;   // Status of Failsafe Digital Input 2
      SS2ESRactive { ExternalWritable := 'False'} : Bool;   // Safety Function SS2ESR active
      SS2Eactive { ExternalWritable := 'False'} : Bool;   // Safety Function SS2E active
      SOSselected { ExternalWritable := 'False'} : Bool;   // Safety Function Safe Operating Stop selected (not active yet)
      SLPupperLimitMaintained { ExternalWritable := 'False'} : Bool;   // SLP: upper limit maintained
      SLPlowerLimitMaintained { ExternalWritable := 'False'} : Bool;   // SLP: lower limit maintained
      SCA1 { ExternalWritable := 'False'} : Bool;   // Safe Cam 1
      SCA2 { ExternalWritable := 'False'} : Bool;   // Safe Cam 2
      SCA3 { ExternalWritable := 'False'} : Bool;   // Safe Cam 3
      SCA4 { ExternalWritable := 'False'} : Bool;   // Safe Cam 4
      SCA5 { ExternalWritable := 'False'} : Bool;   // Safe Cam 5
      SCA6 { ExternalWritable := 'False'} : Bool;   // Safe Cam 6
      SCA7 { ExternalWritable := 'False'} : Bool;   // Safe Cam 7
      SCA8 { ExternalWritable := 'False'} : Bool;   // Safe Cam 8
      SCA9 { ExternalWritable := 'False'} : Bool;   // Safe Cam 9
      SCA10 { ExternalWritable := 'False'} : Bool;   // Safe Cam 10
      SCA11 { ExternalWritable := 'False'} : Bool;   // Safe Cam 11
      SCA12 { ExternalWritable := 'False'} : Bool;   // Safe Cam 12
      SCA13 { ExternalWritable := 'False'} : Bool;   // Safe Cam 13
      SCA14 { ExternalWritable := 'False'} : Bool;   // Safe Cam 14
      SCA15 { ExternalWritable := 'False'} : Bool;   // Safe Cam 15
      SCA16 { ExternalWritable := 'False'} : Bool;   // Safe Cam 16
      SCA17 { ExternalWritable := 'False'} : Bool;   // Safe Cam 17
      SCA18 { ExternalWritable := 'False'} : Bool;   // Safe Cam 18
      SCA19 { ExternalWritable := 'False'} : Bool;   // Safe Cam 19
      SCA20 { ExternalWritable := 'False'} : Bool;   // Safe Cam 20
      SCA21 { ExternalWritable := 'False'} : Bool;   // Safe Cam 21
      SCA22 { ExternalWritable := 'False'} : Bool;   // Safe Cam 22
      SCA23 { ExternalWritable := 'False'} : Bool;   // Safe Cam 23
      SCA24 { ExternalWritable := 'False'} : Bool;   // Safe Cam 24
      SCA25 { ExternalWritable := 'False'} : Bool;   // Safe Cam 25
      SCA26 { ExternalWritable := 'False'} : Bool;   // Safe Cam 26
      SCA27 { ExternalWritable := 'False'} : Bool;   // Safe Cam 27
      SCA28 { ExternalWritable := 'False'} : Bool;   // Safe Cam 28
      SCA29 { ExternalWritable := 'False'} : Bool;   // Safe Cam 29
      SCA30 { ExternalWritable := 'False'} : Bool;   // Safe Cam 30
      SCAactive { ExternalWritable := 'False'} : Bool;   // Safety Function Safe Cam active
      SCAvalid { ExternalWritable := 'False'} : Bool;   // Safety Function Safe Cam valid
      variableSLSvalue { ExternalWritable := 'False'} : Int;   // Actual SLS value for SLS limit 1
   END_STRUCT;
END_TYPE

TYPE "UDT_OPC_ActualValuesAxis"
   STRUCT
      StationNumber : Byte;
      AxisId : DInt;
      ActualPosition : LReal;
   END_STRUCT;
END_TYPE

TYPE "UDT_OPC_Analog"
   STRUCT
      Delay : Real;   // Unit:s
      DiffErrorMax : Real;
      DiffErrorMin : Real;
      DiffWarnMax : Real;
      DiffWarnMin : Real;
      Id : Int;
      Offset : Real;
      Gain : Real := 1.0;
      Target : Real;
      Value : Real;
      Update : Bool;
   END_STRUCT;
END_TYPE

TYPE "UDT_OPC_Button"
   STRUCT
      bBlink : Bool;
      bClick : Bool;
      bEnable : Bool;
      bIsPressed : Bool;
      eColor : Int;   // @Max:4
   END_STRUCT;
END_TYPE

TYPE "UDT_OPC_Maintenance"
   STRUCT
      Elapsed : Real;   // Temps de fonctionnement actuel (en unité de temps)
      Id : Int;   // ID de la tache
      Period : Int;   // Durée maximale avant maintenance
      Reset : Bool;   // Reset Temps de fonctionnement actuel
      WarningThreshold : Int;   // Seuil d'avertissement en % (par défaut 80%)
   END_STRUCT;
END_TYPE

TYPE "UDT_OPC_TaughtPositionsItems"
   STRUCT
      StationNumber : Byte;
      AxisId : DInt;
      PositionId : DInt;
      Value : LReal;
   END_STRUCT;
END_TYPE

TYPE "LBP_typeAlarmMsgs"
TITLE = PLC-Error / Messages / Erreur AP / messages
// User data type for block LBP_AlarmMessage [DB2] / Type de données utilisateur pour bloc LBP_AlarmMessage [DB2]
   STRUCT
      Chan : Array[1..10] of Struct   // From Channel 1..10 / Depuis canal 1..10
         FDD : Array[0..15] of Bool;   // Feed disable / Désactiver avance
         RID : Array[0..15] of Bool;   // Read-in disable / Désactiver importation
         NCSD : Array[0..15] of Bool;   // NC start disable / Désactiver Départ CN
         FdStop_1 : Array[0..15] of Bool;   // Feed stop GEOaxis 1 / Arrêt avance axe GEO 1
         FdStop_2 : Array[0..15] of Bool;   // Feed stop GEOaxis 2 / Arrêt avance axe GEO 2
         FdStop_3 : Array[0..15] of Bool;   // Feed stop GEOaxis 3 / Arrêt avance axe GEO 3
      END_STRUCT;
      Axis : Array[1..31] of Struct   // From Axis 1..31 / Depuis axe 1..31
         FdStop : Array[0..15] of Bool;   // Feed stop axis/spindle / Arrêt avance axe/broche
      END_STRUCT;
      AddValUserA0 : Array[0..63] of Int;   // Additional value for alarms in the user area 0 (700000..700063) / Valeur additionnelle pour les alarmes dans la zone utilisateur 0 (700000..700063)
      ChanA : Array[1..10] of Struct   // From Channel 1..10 / Depuis canal 1..10
         FDD_5C00xx : Array[0..15] of Bool;   // Feed disable Alarm no. 5C0000..5C0015 / Désactiver avance Alarme n° 5C0000..5C0015
         FDD_RID_5C01xx : Array[0..31] of Bool;   // Feed and read-in disable Alarm no. 5C0100..5C0131 / Désactiver avance et importation Alarme n° 5C0100..5C0131
         RID_5C02xx : Array[0..31] of Bool;   // Read-in disable Alarm no. 5C0200..5C0231 / Désactiver avance Alarme n° 5C0200..5C0231
         NCSD_5C03xx : Array[0..15] of Bool;   // NC start disable Alarm no. 5C0300..5C0315 / Désactiver Départ CN Alarme n° 5C0300..5C0315
         FdStop_1_5C11xx : Array[0..15] of Bool;   // Feed stop GEOaxis 1 Alarm no. 5C1100..5C1115 / Arrêt avance axe GEO 1 Alarme n° 5C1100..5C1115
         FdStop_2_5C12xx : Array[0..15] of Bool;   // Feed stop GEOaxis 2 Alarm no. 5C1200..5C1215 / Arrêt avance axe GEO 2 Alarme n° 5C1200..5C1215
         FdStop_3_5C13xx : Array[0..15] of Bool;   // Feed stop GEOaxis 3 Alarm no. 5C1300..5C1315 / Arrêt avance axe GEO 3 Alarme n° 5C1300..5C1315
      END_STRUCT;
      AxisA : Array[1..31] of Struct   // From Axis 1..31 / Depuis axe 1..31
         AAFdStop60AAxx : Array[0..15] of Bool;   // Feed stop axis/spindle / Arrêt avance axe/broche
      END_STRUCT;
      res552 : Word;   // Reserved / Réservé
      UserA : Array[0..63] of Struct
         A70UUxx : Array[0..63] of Bool;   // Alarm 70UU00..70UU63 (user area) / Alarme 70UU00..70UU63 (zone utilisateur)
      END_STRUCT;
   END_STRUCT;
   // // Chan[2].FDD : Feed disable / Désactiver avance
   // // Chan[3].FDD : Feed disable / Désactiver avance
   // // Chan[4].FDD : Feed disable / Désactiver avance
   // // Chan[5].FDD : Feed disable / Désactiver avance
   // // Chan[6].FDD : Feed disable / Désactiver avance
   // // Chan[7].FDD : Feed disable / Désactiver avance
   // // Chan[8].FDD : Feed disable / Désactiver avance
   // // Chan[9].FDD : Feed disable / Désactiver avance
   // // Chan[10].FDD : Feed disable / Désactiver avance
   // // Chan[2].RID : Read-in disable / Désactiver importation
   // // Chan[3].RID : Read-in disable / Désactiver importation
   // // Chan[4].RID : Read-in disable / Désactiver importation
   // // Chan[5].RID : Read-in disable / Désactiver importation
   // // Chan[6].RID : Read-in disable / Désactiver importation
   // // Chan[7].RID : Read-in disable / Désactiver importation
   // // Chan[8].RID : Read-in disable / Désactiver importation
   // // Chan[9].RID : Read-in disable / Désactiver importation
   // // Chan[10].RID : Read-in disable / Désactiver importation
   // // Chan[2].NCSD : NC start disable / Désactiver Départ CN
   // // Chan[3].NCSD : NC start disable / Désactiver Départ CN
   // // Chan[4].NCSD : NC start disable / Désactiver Départ CN
   // // Chan[5].NCSD : NC start disable / Désactiver Départ CN
   // // Chan[6].NCSD : NC start disable / Désactiver Départ CN
   // // Chan[7].NCSD : NC start disable / Désactiver Départ CN
   // // Chan[8].NCSD : NC start disable / Désactiver Départ CN
   // // Chan[9].NCSD : NC start disable / Désactiver Départ CN
   // // Chan[10].NCSD : NC start disable / Désactiver Départ CN
   // // Chan[2].FdStop_1 : Feed stop GEOaxis 1 / Arrêt avance axe GEO 1
   // // Chan[3].FdStop_1 : Feed stop GEOaxis 1 / Arrêt avance axe GEO 1
   // // Chan[4].FdStop_1 : Feed stop GEOaxis 1 / Arrêt avance axe GEO 1
   // // Chan[5].FdStop_1 : Feed stop GEOaxis 1 / Arrêt avance axe GEO 1
   // // Chan[6].FdStop_1 : Feed stop GEOaxis 1 / Arrêt avance axe GEO 1
   // // Chan[7].FdStop_1 : Feed stop GEOaxis 1 / Arrêt avance axe GEO 1
   // // Chan[8].FdStop_1 : Feed stop GEOaxis 1 / Arrêt avance axe GEO 1
   // // Chan[9].FdStop_1 : Feed stop GEOaxis 1 / Arrêt avance axe GEO 1
   // // Chan[10].FdStop_1 : Feed stop GEOaxis 1 / Arrêt avance axe GEO 1
   // // Chan[2].FdStop_2 : Feed stop GEOaxis 2 / Arrêt avance axe GEO 2
   // // Chan[3].FdStop_2 : Feed stop GEOaxis 2 / Arrêt avance axe GEO 2
   // // Chan[4].FdStop_2 : Feed stop GEOaxis 2 / Arrêt avance axe GEO 2
   // // Chan[5].FdStop_2 : Feed stop GEOaxis 2 / Arrêt avance axe GEO 2
   // // Chan[6].FdStop_2 : Feed stop GEOaxis 2 / Arrêt avance axe GEO 2
   // // Chan[7].FdStop_2 : Feed stop GEOaxis 2 / Arrêt avance axe GEO 2
   // // Chan[8].FdStop_2 : Feed stop GEOaxis 2 / Arrêt avance axe GEO 2
   // // Chan[9].FdStop_2 : Feed stop GEOaxis 2 / Arrêt avance axe GEO 2
   // // Chan[10].FdStop_2 : Feed stop GEOaxis 2 / Arrêt avance axe GEO 2
   // // Chan[2].FdStop_3 : Feed stop GEOaxis 3 / Arrêt avance axe GEO 3
   // // Chan[3].FdStop_3 : Feed stop GEOaxis 3 / Arrêt avance axe GEO 3
   // // Chan[4].FdStop_3 : Feed stop GEOaxis 3 / Arrêt avance axe GEO 3
   // // Chan[5].FdStop_3 : Feed stop GEOaxis 3 / Arrêt avance axe GEO 3
   // // Chan[6].FdStop_3 : Feed stop GEOaxis 3 / Arrêt avance axe GEO 3
   // // Chan[7].FdStop_3 : Feed stop GEOaxis 3 / Arrêt avance axe GEO 3
   // // Chan[8].FdStop_3 : Feed stop GEOaxis 3 / Arrêt avance axe GEO 3
   // // Chan[9].FdStop_3 : Feed stop GEOaxis 3 / Arrêt avance axe GEO 3
   // // Chan[10].FdStop_3 : Feed stop GEOaxis 3 / Arrêt avance axe GEO 3
   // // Chan[1] : From Channel 1..10 / Depuis canal 1..10
   // // Chan[2] : From Channel 1..10 / Depuis canal 1..10
   // // Chan[3] : From Channel 1..10 / Depuis canal 1..10
   // // Chan[4] : From Channel 1..10 / Depuis canal 1..10
   // // Chan[5] : From Channel 1..10 / Depuis canal 1..10
   // // Chan[6] : From Channel 1..10 / Depuis canal 1..10
   // // Chan[7] : From Channel 1..10 / Depuis canal 1..10
   // // Chan[8] : From Channel 1..10 / Depuis canal 1..10
   // // Chan[9] : From Channel 1..10 / Depuis canal 1..10
   // // Chan[10] : From Channel 1..10 / Depuis canal 1..10
   // // Axis[2].FdStop : Feed stop axis/spindle / Arrêt avance axe/broche
   // // Axis[3].FdStop : Feed stop axis/spindle / Arrêt avance axe/broche
   // // Axis[4].FdStop : Feed stop axis/spindle / Arrêt avance axe/broche
   // // Axis[5].FdStop : Feed stop axis/spindle / Arrêt avance axe/broche
   // // Axis[6].FdStop : Feed stop axis/spindle / Arrêt avance axe/broche
   // // Axis[7].FdStop : Feed stop axis/spindle / Arrêt avance axe/broche
   // // Axis[8].FdStop : Feed stop axis/spindle / Arrêt avance axe/broche
   // // Axis[9].FdStop : Feed stop axis/spindle / Arrêt avance axe/broche
   // // Axis[10].FdStop : Feed stop axis/spindle / Arrêt avance axe/broche
   // // Axis[11].FdStop : Feed stop axis/spindle / Arrêt avance axe/broche
   // // Axis[12].FdStop : Feed stop axis/spindle / Arrêt avance axe/broche
   // // Axis[13].FdStop : Feed stop axis/spindle / Arrêt avance axe/broche
   // // Axis[14].FdStop : Feed stop axis/spindle / Arrêt avance axe/broche
   // // Axis[15].FdStop : Feed stop axis/spindle / Arrêt avance axe/broche
   // // Axis[16].FdStop : Feed stop axis/spindle / Arrêt avance axe/broche
   // // Axis[17].FdStop : Feed stop axis/spindle / Arrêt avance axe/broche
   // // Axis[18].FdStop : Feed stop axis/spindle / Arrêt avance axe/broche
   // // Axis[19].FdStop : Feed stop axis/spindle / Arrêt avance axe/broche
   // // Axis[20].FdStop : Feed stop axis/spindle / Arrêt avance axe/broche
   // // Axis[21].FdStop : Feed stop axis/spindle / Arrêt avance axe/broche
   // // Axis[22].FdStop : Feed stop axis/spindle / Arrêt avance axe/broche
   // // Axis[23].FdStop : Feed stop axis/spindle / Arrêt avance axe/broche
   // // Axis[24].FdStop : Feed stop axis/spindle / Arrêt avance axe/broche
   // // Axis[25].FdStop : Feed stop axis/spindle / Arrêt avance axe/broche
   // // Axis[26].FdStop : Feed stop axis/spindle / Arrêt avance axe/broche
   // // Axis[27].FdStop : Feed stop axis/spindle / Arrêt avance axe/broche
   // // Axis[28].FdStop : Feed stop axis/spindle / Arrêt avance axe/broche
   // // Axis[29].FdStop : Feed stop axis/spindle / Arrêt avance axe/broche
   // // Axis[30].FdStop : Feed stop axis/spindle / Arrêt avance axe/broche
   // // Axis[31].FdStop : Feed stop axis/spindle / Arrêt avance axe/broche
   // // Axis[1] : From Axis 1..31 / Depuis axe 1..31
   // // Axis[2] : From Axis 1..31 / Depuis axe 1..31
   // // Axis[3] : From Axis 1..31 / Depuis axe 1..31
   // // Axis[4] : From Axis 1..31 / Depuis axe 1..31
   // // Axis[5] : From Axis 1..31 / Depuis axe 1..31
   // // Axis[6] : From Axis 1..31 / Depuis axe 1..31
   // // Axis[7] : From Axis 1..31 / Depuis axe 1..31
   // // Axis[8] : From Axis 1..31 / Depuis axe 1..31
   // // Axis[9] : From Axis 1..31 / Depuis axe 1..31
   // // Axis[10] : From Axis 1..31 / Depuis axe 1..31
   // // Axis[11] : From Axis 1..31 / Depuis axe 1..31
   // // Axis[12] : From Axis 1..31 / Depuis axe 1..31
   // // Axis[13] : From Axis 1..31 / Depuis axe 1..31
   // // Axis[14] : From Axis 1..31 / Depuis axe 1..31
   // // Axis[15] : From Axis 1..31 / Depuis axe 1..31
   // // Axis[16] : From Axis 1..31 / Depuis axe 1..31
   // // Axis[17] : From Axis 1..31 / Depuis axe 1..31
   // // Axis[18] : From Axis 1..31 / Depuis axe 1..31
   // // Axis[19] : From Axis 1..31 / Depuis axe 1..31
   // // Axis[20] : From Axis 1..31 / Depuis axe 1..31
   // // Axis[21] : From Axis 1..31 / Depuis axe 1..31
   // // Axis[22] : From Axis 1..31 / Depuis axe 1..31
   // // Axis[23] : From Axis 1..31 / Depuis axe 1..31
   // // Axis[24] : From Axis 1..31 / Depuis axe 1..31
   // // Axis[25] : From Axis 1..31 / Depuis axe 1..31
   // // Axis[26] : From Axis 1..31 / Depuis axe 1..31
   // // Axis[27] : From Axis 1..31 / Depuis axe 1..31
   // // Axis[28] : From Axis 1..31 / Depuis axe 1..31
   // // Axis[29] : From Axis 1..31 / Depuis axe 1..31
   // // Axis[30] : From Axis 1..31 / Depuis axe 1..31
   // // Axis[31] : From Axis 1..31 / Depuis axe 1..31
   // // ChanA[2].FDD_5C00xx : Feed disable Alarm no. 5C0000..5C0015 / Désactiver avance Alarme n° 5C0000..5C0015
   // // ChanA[3].FDD_5C00xx : Feed disable Alarm no. 5C0000..5C0015 / Désactiver avance Alarme n° 5C0000..5C0015
   // // ChanA[4].FDD_5C00xx : Feed disable Alarm no. 5C0000..5C0015 / Désactiver avance Alarme n° 5C0000..5C0015
   // // ChanA[5].FDD_5C00xx : Feed disable Alarm no. 5C0000..5C0015 / Désactiver avance Alarme n° 5C0000..5C0015
   // // ChanA[6].FDD_5C00xx : Feed disable Alarm no. 5C0000..5C0015 / Désactiver avance Alarme n° 5C0000..5C0015
   // // ChanA[7].FDD_5C00xx : Feed disable Alarm no. 5C0000..5C0015 / Désactiver avance Alarme n° 5C0000..5C0015
   // // ChanA[8].FDD_5C00xx : Feed disable Alarm no. 5C0000..5C0015 / Désactiver avance Alarme n° 5C0000..5C0015
   // // ChanA[9].FDD_5C00xx : Feed disable Alarm no. 5C0000..5C0015 / Désactiver avance Alarme n° 5C0000..5C0015
   // // ChanA[10].FDD_5C00xx : Feed disable Alarm no. 5C0000..5C0015 / Désactiver avance Alarme n° 5C0000..5C0015
   // // ChanA[2].FDD_RID_5C01xx : Feed and read-in disable Alarm no. 5C0100..5C0131 / Désactiver avance et importation Alarme n° 5C0100..5C0131
   // // ChanA[3].FDD_RID_5C01xx : Feed and read-in disable Alarm no. 5C0100..5C0131 / Désactiver avance et importation Alarme n° 5C0100..5C0131
   // // ChanA[4].FDD_RID_5C01xx : Feed and read-in disable Alarm no. 5C0100..5C0131 / Désactiver avance et importation Alarme n° 5C0100..5C0131
   // // ChanA[5].FDD_RID_5C01xx : Feed and read-in disable Alarm no. 5C0100..5C0131 / Désactiver avance et importation Alarme n° 5C0100..5C0131
   // // ChanA[6].FDD_RID_5C01xx : Feed and read-in disable Alarm no. 5C0100..5C0131 / Désactiver avance et importation Alarme n° 5C0100..5C0131
   // // ChanA[7].FDD_RID_5C01xx : Feed and read-in disable Alarm no. 5C0100..5C0131 / Désactiver avance et importation Alarme n° 5C0100..5C0131
   // // ChanA[8].FDD_RID_5C01xx : Feed and read-in disable Alarm no. 5C0100..5C0131 / Désactiver avance et importation Alarme n° 5C0100..5C0131
   // // ChanA[9].FDD_RID_5C01xx : Feed and read-in disable Alarm no. 5C0100..5C0131 / Désactiver avance et importation Alarme n° 5C0100..5C0131
   // // ChanA[10].FDD_RID_5C01xx : Feed and read-in disable Alarm no. 5C0100..5C0131 / Désactiver avance et importation Alarme n° 5C0100..5C0131
   // // ChanA[2].RID_5C02xx : Read-in disable Alarm no. 5C0200..5C0231 / Désactiver avance Alarme n° 5C0200..5C0231
   // // ChanA[3].RID_5C02xx : Read-in disable Alarm no. 5C0200..5C0231 / Désactiver avance Alarme n° 5C0200..5C0231
   // // ChanA[4].RID_5C02xx : Read-in disable Alarm no. 5C0200..5C0231 / Désactiver avance Alarme n° 5C0200..5C0231
   // // ChanA[5].RID_5C02xx : Read-in disable Alarm no. 5C0200..5C0231 / Désactiver avance Alarme n° 5C0200..5C0231
   // // ChanA[6].RID_5C02xx : Read-in disable Alarm no. 5C0200..5C0231 / Désactiver avance Alarme n° 5C0200..5C0231
   // // ChanA[7].RID_5C02xx : Read-in disable Alarm no. 5C0200..5C0231 / Désactiver avance Alarme n° 5C0200..5C0231
   // // ChanA[8].RID_5C02xx : Read-in disable Alarm no. 5C0200..5C0231 / Désactiver avance Alarme n° 5C0200..5C0231
   // // ChanA[9].RID_5C02xx : Read-in disable Alarm no. 5C0200..5C0231 / Désactiver avance Alarme n° 5C0200..5C0231
   // // ChanA[10].RID_5C02xx : Read-in disable Alarm no. 5C0200..5C0231 / Désactiver avance Alarme n° 5C0200..5C0231
   // // ChanA[2].NCSD_5C03xx : NC start disable Alarm no. 5C0300..5C0315 / Désactiver Départ CN Alarme n° 5C0300..5C0315
   // // ChanA[3].NCSD_5C03xx : NC start disable Alarm no. 5C0300..5C0315 / Désactiver Départ CN Alarme n° 5C0300..5C0315
   // // ChanA[4].NCSD_5C03xx : NC start disable Alarm no. 5C0300..5C0315 / Désactiver Départ CN Alarme n° 5C0300..5C0315
   // // ChanA[5].NCSD_5C03xx : NC start disable Alarm no. 5C0300..5C0315 / Désactiver Départ CN Alarme n° 5C0300..5C0315
   // // ChanA[6].NCSD_5C03xx : NC start disable Alarm no. 5C0300..5C0315 / Désactiver Départ CN Alarme n° 5C0300..5C0315
   // // ChanA[7].NCSD_5C03xx : NC start disable Alarm no. 5C0300..5C0315 / Désactiver Départ CN Alarme n° 5C0300..5C0315
   // // ChanA[8].NCSD_5C03xx : NC start disable Alarm no. 5C0300..5C0315 / Désactiver Départ CN Alarme n° 5C0300..5C0315
   // // ChanA[9].NCSD_5C03xx : NC start disable Alarm no. 5C0300..5C0315 / Désactiver Départ CN Alarme n° 5C0300..5C0315
   // // ChanA[10].NCSD_5C03xx : NC start disable Alarm no. 5C0300..5C0315 / Désactiver Départ CN Alarme n° 5C0300..5C0315
   // // ChanA[2].FdStop_1_5C11xx : Feed stop GEOaxis 1 Alarm no. 5C1100..5C1115 / Arrêt avance axe GEO 1 Alarme n° 5C1100..5C1115
   // // ChanA[3].FdStop_1_5C11xx : Feed stop GEOaxis 1 Alarm no. 5C1100..5C1115 / Arrêt avance axe GEO 1 Alarme n° 5C1100..5C1115
   // // ChanA[4].FdStop_1_5C11xx : Feed stop GEOaxis 1 Alarm no. 5C1100..5C1115 / Arrêt avance axe GEO 1 Alarme n° 5C1100..5C1115
   // // ChanA[5].FdStop_1_5C11xx : Feed stop GEOaxis 1 Alarm no. 5C1100..5C1115 / Arrêt avance axe GEO 1 Alarme n° 5C1100..5C1115
   // // ChanA[6].FdStop_1_5C11xx : Feed stop GEOaxis 1 Alarm no. 5C1100..5C1115 / Arrêt avance axe GEO 1 Alarme n° 5C1100..5C1115
   // // ChanA[7].FdStop_1_5C11xx : Feed stop GEOaxis 1 Alarm no. 5C1100..5C1115 / Arrêt avance axe GEO 1 Alarme n° 5C1100..5C1115
   // // ChanA[8].FdStop_1_5C11xx : Feed stop GEOaxis 1 Alarm no. 5C1100..5C1115 / Arrêt avance axe GEO 1 Alarme n° 5C1100..5C1115
   // // ChanA[9].FdStop_1_5C11xx : Feed stop GEOaxis 1 Alarm no. 5C1100..5C1115 / Arrêt avance axe GEO 1 Alarme n° 5C1100..5C1115
   // // ChanA[10].FdStop_1_5C11xx : Feed stop GEOaxis 1 Alarm no. 5C1100..5C1115 / Arrêt avance axe GEO 1 Alarme n° 5C1100..5C1115
   // // ChanA[2].FdStop_2_5C12xx : Feed stop GEOaxis 2 Alarm no. 5C1200..5C1215 / Arrêt avance axe GEO 2 Alarme n° 5C1200..5C1215
   // // ChanA[3].FdStop_2_5C12xx : Feed stop GEOaxis 2 Alarm no. 5C1200..5C1215 / Arrêt avance axe GEO 2 Alarme n° 5C1200..5C1215
   // // ChanA[4].FdStop_2_5C12xx : Feed stop GEOaxis 2 Alarm no. 5C1200..5C1215 / Arrêt avance axe GEO 2 Alarme n° 5C1200..5C1215
   // // ChanA[5].FdStop_2_5C12xx : Feed stop GEOaxis 2 Alarm no. 5C1200..5C1215 / Arrêt avance axe GEO 2 Alarme n° 5C1200..5C1215
   // // ChanA[6].FdStop_2_5C12xx : Feed stop GEOaxis 2 Alarm no. 5C1200..5C1215 / Arrêt avance axe GEO 2 Alarme n° 5C1200..5C1215
   // // ChanA[7].FdStop_2_5C12xx : Feed stop GEOaxis 2 Alarm no. 5C1200..5C1215 / Arrêt avance axe GEO 2 Alarme n° 5C1200..5C1215
   // // ChanA[8].FdStop_2_5C12xx : Feed stop GEOaxis 2 Alarm no. 5C1200..5C1215 / Arrêt avance axe GEO 2 Alarme n° 5C1200..5C1215
   // // ChanA[9].FdStop_2_5C12xx : Feed stop GEOaxis 2 Alarm no. 5C1200..5C1215 / Arrêt avance axe GEO 2 Alarme n° 5C1200..5C1215
   // // ChanA[10].FdStop_2_5C12xx : Feed stop GEOaxis 2 Alarm no. 5C1200..5C1215 / Arrêt avance axe GEO 2 Alarme n° 5C1200..5C1215
   // // ChanA[2].FdStop_3_5C13xx : Feed stop GEOaxis 3 Alarm no. 5C1300..5C1315 / Arrêt avance axe GEO 3 Alarme n° 5C1300..5C1315
   // // ChanA[3].FdStop_3_5C13xx : Feed stop GEOaxis 3 Alarm no. 5C1300..5C1315 / Arrêt avance axe GEO 3 Alarme n° 5C1300..5C1315
   // // ChanA[4].FdStop_3_5C13xx : Feed stop GEOaxis 3 Alarm no. 5C1300..5C1315 / Arrêt avance axe GEO 3 Alarme n° 5C1300..5C1315
   // // ChanA[5].FdStop_3_5C13xx : Feed stop GEOaxis 3 Alarm no. 5C1300..5C1315 / Arrêt avance axe GEO 3 Alarme n° 5C1300..5C1315
   // // ChanA[6].FdStop_3_5C13xx : Feed stop GEOaxis 3 Alarm no. 5C1300..5C1315 / Arrêt avance axe GEO 3 Alarme n° 5C1300..5C1315
   // // ChanA[7].FdStop_3_5C13xx : Feed stop GEOaxis 3 Alarm no. 5C1300..5C1315 / Arrêt avance axe GEO 3 Alarme n° 5C1300..5C1315
   // // ChanA[8].FdStop_3_5C13xx : Feed stop GEOaxis 3 Alarm no. 5C1300..5C1315 / Arrêt avance axe GEO 3 Alarme n° 5C1300..5C1315
   // // ChanA[9].FdStop_3_5C13xx : Feed stop GEOaxis 3 Alarm no. 5C1300..5C1315 / Arrêt avance axe GEO 3 Alarme n° 5C1300..5C1315
   // // ChanA[10].FdStop_3_5C13xx : Feed stop GEOaxis 3 Alarm no. 5C1300..5C1315 / Arrêt avance axe GEO 3 Alarme n° 5C1300..5C1315
   // // ChanA[1] : From Channel 1..10 / Depuis canal 1..10
   // // ChanA[2] : From Channel 1..10 / Depuis canal 1..10
   // // ChanA[3] : From Channel 1..10 / Depuis canal 1..10
   // // ChanA[4] : From Channel 1..10 / Depuis canal 1..10
   // // ChanA[5] : From Channel 1..10 / Depuis canal 1..10
   // // ChanA[6] : From Channel 1..10 / Depuis canal 1..10
   // // ChanA[7] : From Channel 1..10 / Depuis canal 1..10
   // // ChanA[8] : From Channel 1..10 / Depuis canal 1..10
   // // ChanA[9] : From Channel 1..10 / Depuis canal 1..10
   // // ChanA[10] : From Channel 1..10 / Depuis canal 1..10
   // // AxisA[2].AAFdStop60AAxx : Feed stop axis/spindle / Arrêt avance axe/broche
   // // AxisA[3].AAFdStop60AAxx : Feed stop axis/spindle / Arrêt avance axe/broche
   // // AxisA[4].AAFdStop60AAxx : Feed stop axis/spindle / Arrêt avance axe/broche
   // // AxisA[5].AAFdStop60AAxx : Feed stop axis/spindle / Arrêt avance axe/broche
   // // AxisA[6].AAFdStop60AAxx : Feed stop axis/spindle / Arrêt avance axe/broche
   // // AxisA[7].AAFdStop60AAxx : Feed stop axis/spindle / Arrêt avance axe/broche
   // // AxisA[8].AAFdStop60AAxx : Feed stop axis/spindle / Arrêt avance axe/broche
   // // AxisA[9].AAFdStop60AAxx : Feed stop axis/spindle / Arrêt avance axe/broche
   // // AxisA[10].AAFdStop60AAxx : Feed stop axis/spindle / Arrêt avance axe/broche
   // // AxisA[11].AAFdStop60AAxx : Feed stop axis/spindle / Arrêt avance axe/broche
   // // AxisA[12].AAFdStop60AAxx : Feed stop axis/spindle / Arrêt avance axe/broche
   // // AxisA[13].AAFdStop60AAxx : Feed stop axis/spindle / Arrêt avance axe/broche
   // // AxisA[14].AAFdStop60AAxx : Feed stop axis/spindle / Arrêt avance axe/broche
   // // AxisA[15].AAFdStop60AAxx : Feed stop axis/spindle / Arrêt avance axe/broche
   // // AxisA[16].AAFdStop60AAxx : Feed stop axis/spindle / Arrêt avance axe/broche
   // // AxisA[17].AAFdStop60AAxx : Feed stop axis/spindle / Arrêt avance axe/broche
   // // AxisA[18].AAFdStop60AAxx : Feed stop axis/spindle / Arrêt avance axe/broche
   // // AxisA[19].AAFdStop60AAxx : Feed stop axis/spindle / Arrêt avance axe/broche
   // // AxisA[20].AAFdStop60AAxx : Feed stop axis/spindle / Arrêt avance axe/broche
   // // AxisA[21].AAFdStop60AAxx : Feed stop axis/spindle / Arrêt avance axe/broche
   // // AxisA[22].AAFdStop60AAxx : Feed stop axis/spindle / Arrêt avance axe/broche
   // // AxisA[23].AAFdStop60AAxx : Feed stop axis/spindle / Arrêt avance axe/broche
   // // AxisA[24].AAFdStop60AAxx : Feed stop axis/spindle / Arrêt avance axe/broche
   // // AxisA[25].AAFdStop60AAxx : Feed stop axis/spindle / Arrêt avance axe/broche
   // // AxisA[26].AAFdStop60AAxx : Feed stop axis/spindle / Arrêt avance axe/broche
   // // AxisA[27].AAFdStop60AAxx : Feed stop axis/spindle / Arrêt avance axe/broche
   // // AxisA[28].AAFdStop60AAxx : Feed stop axis/spindle / Arrêt avance axe/broche
   // // AxisA[29].AAFdStop60AAxx : Feed stop axis/spindle / Arrêt avance axe/broche
   // // AxisA[30].AAFdStop60AAxx : Feed stop axis/spindle / Arrêt avance axe/broche
   // // AxisA[31].AAFdStop60AAxx : Feed stop axis/spindle / Arrêt avance axe/broche
   // // AxisA[1] : From Axis 1..31 / Depuis axe 1..31
   // // AxisA[2] : From Axis 1..31 / Depuis axe 1..31
   // // AxisA[3] : From Axis 1..31 / Depuis axe 1..31
   // // AxisA[4] : From Axis 1..31 / Depuis axe 1..31
   // // AxisA[5] : From Axis 1..31 / Depuis axe 1..31
   // // AxisA[6] : From Axis 1..31 / Depuis axe 1..31
   // // AxisA[7] : From Axis 1..31 / Depuis axe 1..31
   // // AxisA[8] : From Axis 1..31 / Depuis axe 1..31
   // // AxisA[9] : From Axis 1..31 / Depuis axe 1..31
   // // AxisA[10] : From Axis 1..31 / Depuis axe 1..31
   // // AxisA[11] : From Axis 1..31 / Depuis axe 1..31
   // // AxisA[12] : From Axis 1..31 / Depuis axe 1..31
   // // AxisA[13] : From Axis 1..31 / Depuis axe 1..31
   // // AxisA[14] : From Axis 1..31 / Depuis axe 1..31
   // // AxisA[15] : From Axis 1..31 / Depuis axe 1..31
   // // AxisA[16] : From Axis 1..31 / Depuis axe 1..31
   // // AxisA[17] : From Axis 1..31 / Depuis axe 1..31
   // // AxisA[18] : From Axis 1..31 / Depuis axe 1..31
   // // AxisA[19] : From Axis 1..31 / Depuis axe 1..31
   // // AxisA[20] : From Axis 1..31 / Depuis axe 1..31
   // // AxisA[21] : From Axis 1..31 / Depuis axe 1..31
   // // AxisA[22] : From Axis 1..31 / Depuis axe 1..31
   // // AxisA[23] : From Axis 1..31 / Depuis axe 1..31
   // // AxisA[24] : From Axis 1..31 / Depuis axe 1..31
   // // AxisA[25] : From Axis 1..31 / Depuis axe 1..31
   // // AxisA[26] : From Axis 1..31 / Depuis axe 1..31
   // // AxisA[27] : From Axis 1..31 / Depuis axe 1..31
   // // AxisA[28] : From Axis 1..31 / Depuis axe 1..31
   // // AxisA[29] : From Axis 1..31 / Depuis axe 1..31
   // // AxisA[30] : From Axis 1..31 / Depuis axe 1..31
   // // AxisA[31] : From Axis 1..31 / Depuis axe 1..31
   // // UserA[1].A70UUxx : Alarm 70UU00..70UU63 (user area) / Alarme 70UU00..70UU63 (zone utilisateur)
   // // UserA[2].A70UUxx : Alarm 70UU00..70UU63 (user area) / Alarme 70UU00..70UU63 (zone utilisateur)
   // // UserA[3].A70UUxx : Alarm 70UU00..70UU63 (user area) / Alarme 70UU00..70UU63 (zone utilisateur)
   // // UserA[4].A70UUxx : Alarm 70UU00..70UU63 (user area) / Alarme 70UU00..70UU63 (zone utilisateur)
   // // UserA[5].A70UUxx : Alarm 70UU00..70UU63 (user area) / Alarme 70UU00..70UU63 (zone utilisateur)
   // // UserA[6].A70UUxx : Alarm 70UU00..70UU63 (user area) / Alarme 70UU00..70UU63 (zone utilisateur)
   // // UserA[7].A70UUxx : Alarm 70UU00..70UU63 (user area) / Alarme 70UU00..70UU63 (zone utilisateur)
   // // UserA[8].A70UUxx : Alarm 70UU00..70UU63 (user area) / Alarme 70UU00..70UU63 (zone utilisateur)
   // // UserA[9].A70UUxx : Alarm 70UU00..70UU63 (user area) / Alarme 70UU00..70UU63 (zone utilisateur)
   // // UserA[10].A70UUxx : Alarm 70UU00..70UU63 (user area) / Alarme 70UU00..70UU63 (zone utilisateur)
   // // UserA[11].A70UUxx : Alarm 70UU00..70UU63 (user area) / Alarme 70UU00..70UU63 (zone utilisateur)
   // // UserA[12].A70UUxx : Alarm 70UU00..70UU63 (user area) / Alarme 70UU00..70UU63 (zone utilisateur)
   // // UserA[13].A70UUxx : Alarm 70UU00..70UU63 (user area) / Alarme 70UU00..70UU63 (zone utilisateur)
   // // UserA[14].A70UUxx : Alarm 70UU00..70UU63 (user area) / Alarme 70UU00..70UU63 (zone utilisateur)
   // // UserA[15].A70UUxx : Alarm 70UU00..70UU63 (user area) / Alarme 70UU00..70UU63 (zone utilisateur)
   // // UserA[16].A70UUxx : Alarm 70UU00..70UU63 (user area) / Alarme 70UU00..70UU63 (zone utilisateur)
   // // UserA[17].A70UUxx : Alarm 70UU00..70UU63 (user area) / Alarme 70UU00..70UU63 (zone utilisateur)
   // // UserA[18].A70UUxx : Alarm 70UU00..70UU63 (user area) / Alarme 70UU00..70UU63 (zone utilisateur)
   // // UserA[19].A70UUxx : Alarm 70UU00..70UU63 (user area) / Alarme 70UU00..70UU63 (zone utilisateur)
   // // UserA[20].A70UUxx : Alarm 70UU00..70UU63 (user area) / Alarme 70UU00..70UU63 (zone utilisateur)
   // // UserA[21].A70UUxx : Alarm 70UU00..70UU63 (user area) / Alarme 70UU00..70UU63 (zone utilisateur)
   // // UserA[22].A70UUxx : Alarm 70UU00..70UU63 (user area) / Alarme 70UU00..70UU63 (zone utilisateur)
   // // UserA[23].A70UUxx : Alarm 70UU00..70UU63 (user area) / Alarme 70UU00..70UU63 (zone utilisateur)
   // // UserA[24].A70UUxx : Alarm 70UU00..70UU63 (user area) / Alarme 70UU00..70UU63 (zone utilisateur)
   // // UserA[25].A70UUxx : Alarm 70UU00..70UU63 (user area) / Alarme 70UU00..70UU63 (zone utilisateur)
   // // UserA[26].A70UUxx : Alarm 70UU00..70UU63 (user area) / Alarme 70UU00..70UU63 (zone utilisateur)
   // // UserA[27].A70UUxx : Alarm 70UU00..70UU63 (user area) / Alarme 70UU00..70UU63 (zone utilisateur)
   // // UserA[28].A70UUxx : Alarm 70UU00..70UU63 (user area) / Alarme 70UU00..70UU63 (zone utilisateur)
   // // UserA[29].A70UUxx : Alarm 70UU00..70UU63 (user area) / Alarme 70UU00..70UU63 (zone utilisateur)
   // // UserA[30].A70UUxx : Alarm 70UU00..70UU63 (user area) / Alarme 70UU00..70UU63 (zone utilisateur)
   // // UserA[31].A70UUxx : Alarm 70UU00..70UU63 (user area) / Alarme 70UU00..70UU63 (zone utilisateur)
   // // UserA[32].A70UUxx : Alarm 70UU00..70UU63 (user area) / Alarme 70UU00..70UU63 (zone utilisateur)
   // // UserA[33].A70UUxx : Alarm 70UU00..70UU63 (user area) / Alarme 70UU00..70UU63 (zone utilisateur)
   // // UserA[34].A70UUxx : Alarm 70UU00..70UU63 (user area) / Alarme 70UU00..70UU63 (zone utilisateur)
   // // UserA[35].A70UUxx : Alarm 70UU00..70UU63 (user area) / Alarme 70UU00..70UU63 (zone utilisateur)
   // // UserA[36].A70UUxx : Alarm 70UU00..70UU63 (user area) / Alarme 70UU00..70UU63 (zone utilisateur)
   // // UserA[37].A70UUxx : Alarm 70UU00..70UU63 (user area) / Alarme 70UU00..70UU63 (zone utilisateur)
   // // UserA[38].A70UUxx : Alarm 70UU00..70UU63 (user area) / Alarme 70UU00..70UU63 (zone utilisateur)
   // // UserA[39].A70UUxx : Alarm 70UU00..70UU63 (user area) / Alarme 70UU00..70UU63 (zone utilisateur)
   // // UserA[40].A70UUxx : Alarm 70UU00..70UU63 (user area) / Alarme 70UU00..70UU63 (zone utilisateur)
   // // UserA[41].A70UUxx : Alarm 70UU00..70UU63 (user area) / Alarme 70UU00..70UU63 (zone utilisateur)
   // // UserA[42].A70UUxx : Alarm 70UU00..70UU63 (user area) / Alarme 70UU00..70UU63 (zone utilisateur)
   // // UserA[43].A70UUxx : Alarm 70UU00..70UU63 (user area) / Alarme 70UU00..70UU63 (zone utilisateur)
   // // UserA[44].A70UUxx : Alarm 70UU00..70UU63 (user area) / Alarme 70UU00..70UU63 (zone utilisateur)
   // // UserA[45].A70UUxx : Alarm 70UU00..70UU63 (user area) / Alarme 70UU00..70UU63 (zone utilisateur)
   // // UserA[46].A70UUxx : Alarm 70UU00..70UU63 (user area) / Alarme 70UU00..70UU63 (zone utilisateur)
   // // UserA[47].A70UUxx : Alarm 70UU00..70UU63 (user area) / Alarme 70UU00..70UU63 (zone utilisateur)
   // // UserA[48].A70UUxx : Alarm 70UU00..70UU63 (user area) / Alarme 70UU00..70UU63 (zone utilisateur)
   // // UserA[49].A70UUxx : Alarm 70UU00..70UU63 (user area) / Alarme 70UU00..70UU63 (zone utilisateur)
   // // UserA[50].A70UUxx : Alarm 70UU00..70UU63 (user area) / Alarme 70UU00..70UU63 (zone utilisateur)
   // // UserA[51].A70UUxx : Alarm 70UU00..70UU63 (user area) / Alarme 70UU00..70UU63 (zone utilisateur)
   // // UserA[52].A70UUxx : Alarm 70UU00..70UU63 (user area) / Alarme 70UU00..70UU63 (zone utilisateur)
   // // UserA[53].A70UUxx : Alarm 70UU00..70UU63 (user area) / Alarme 70UU00..70UU63 (zone utilisateur)
   // // UserA[54].A70UUxx : Alarm 70UU00..70UU63 (user area) / Alarme 70UU00..70UU63 (zone utilisateur)
   // // UserA[55].A70UUxx : Alarm 70UU00..70UU63 (user area) / Alarme 70UU00..70UU63 (zone utilisateur)
   // // UserA[56].A70UUxx : Alarm 70UU00..70UU63 (user area) / Alarme 70UU00..70UU63 (zone utilisateur)
   // // UserA[57].A70UUxx : Alarm 70UU00..70UU63 (user area) / Alarme 70UU00..70UU63 (zone utilisateur)
   // // UserA[58].A70UUxx : Alarm 70UU00..70UU63 (user area) / Alarme 70UU00..70UU63 (zone utilisateur)
   // // UserA[59].A70UUxx : Alarm 70UU00..70UU63 (user area) / Alarme 70UU00..70UU63 (zone utilisateur)
   // // UserA[60].A70UUxx : Alarm 70UU00..70UU63 (user area) / Alarme 70UU00..70UU63 (zone utilisateur)
   // // UserA[61].A70UUxx : Alarm 70UU00..70UU63 (user area) / Alarme 70UU00..70UU63 (zone utilisateur)
   // // UserA[62].A70UUxx : Alarm 70UU00..70UU63 (user area) / Alarme 70UU00..70UU63 (zone utilisateur)
   // // UserA[63].A70UUxx : Alarm 70UU00..70UU63 (user area) / Alarme 70UU00..70UU63 (zone utilisateur)
END_TYPE

